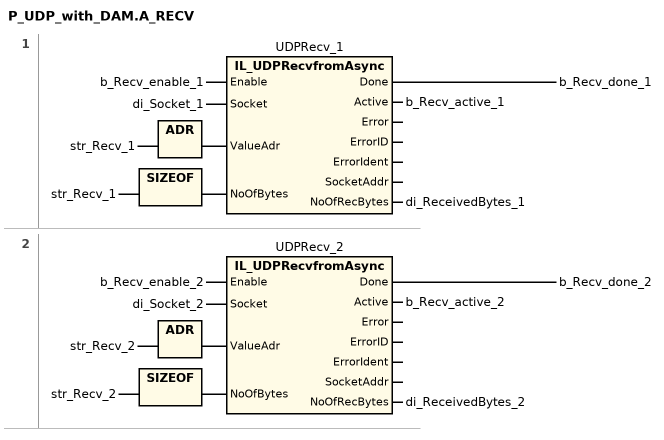
// NETWORK 1
UDPRecv_1(
    Enable := b_Recv_enable_1,
    Socket := di_Socket_1,
    ValueAdr := ADR(str_Recv_1),
    NoOfBytes := SIZEOF(str_Recv_1),
    Active => b_Recv_active_1,
    NoOfRecBytes => di_ReceivedBytes_1); // IL_UDPRecvfromAsync
b_Recv_done_1 := UDPRecv_1.Done;

// NETWORK 2
UDPRecv_2(
    Enable := b_Recv_enable_2,
    Socket := di_Socket_2,
    ValueAdr := ADR(str_Recv_2),
    NoOfBytes := SIZEOF(str_Recv_2),
    Active => b_Recv_active_2,
    NoOfRecBytes => di_ReceivedBytes_2); // IL_UDPRecvfromAsync
b_Recv_done_2 := UDPRecv_2.Done;
END_ACTION

ACTION A_SEND:
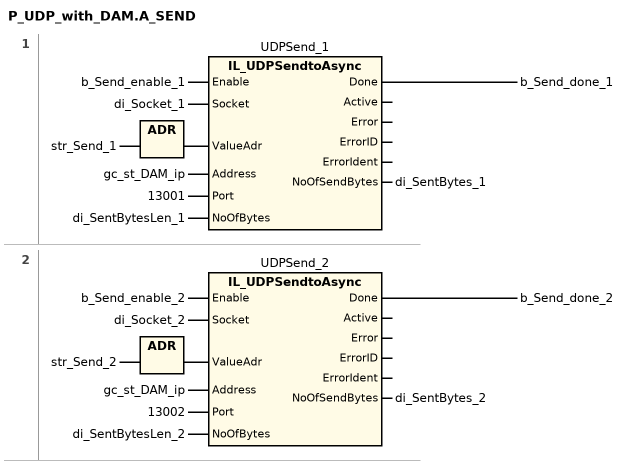
// NETWORK 1
UDPSend_1(
    Enable := b_Send_enable_1,
    Socket := di_Socket_1,
    ValueAdr := ADR(str_Send_1),
    Address := gc_st_DAM_ip,
    Port := 13001,
    NoOfBytes := di_SentBytesLen_1,
    NoOfSendBytes => di_SentBytes_1); // IL_UDPSendtoAsync
b_Send_done_1 := UDPSend_1.Done;

// NETWORK 2
UDPSend_2(
    Enable := b_Send_enable_2,
    Socket := di_Socket_2,
    ValueAdr := ADR(str_Send_2),
    Address := gc_st_DAM_ip,
    Port := 13002,
    NoOfBytes := di_SentBytesLen_2,
    NoOfSendBytes => di_SentBytes_2); // IL_UDPSendtoAsync
b_Send_done_2 := UDPSend_2.Done;
END_ACTION

END_PROGRAM

// IndraMotionMlc1/Application/POUs/TCP/Message/CRC16_MODBUS
FUNCTION_BLOCK CRC16_MODBUS
VAR_INPUT
	str_Message: ARRAY[1..40] OF BYTE;
	str_Len: BYTE;
END_VAR
VAR_OUTPUT
	crc16 : WORD;
END_VAR
VAR
	i : BYTE;
	j : BYTE;
	polynomial : WORD;
	curval : WORD;
	temp : WORD;
END_VAR


temp := 16#FFFF;
polynomial := 16#A001;
FOR i:=1 TO str_Len BY 1 DO
	curval := BYTE_TO_WORD(str_Message[i]);
	FOR j:=1 TO 8 BY 1 DO
		IF ((WORD_TO_BYTE(temp XOR curval) AND 16#01) = 16#01) THEN
			temp := (SHR(temp,1) XOR polynomial);
		ELSE
			temp := SHR(temp,1);			
		END_IF;
		curval := SHR(curval,1);
	END_FOR;
END_FOR;

crc16 := temp;

END_FUNCTION_BLOCK

// IndraMotionMlc1/Application/POUs/TCP/P_GSTAT_K2STAT
(*the program is built for GSTAT and KSTAT,according to ICD*)
PROGRAM P_GSTAT_K2STAT
VAR
(*the transitional variables for GSTAT and KSTAT*)
    STR_GSTAT: STRING(1500);
	STR_K2STAT: STRING(255);
	STR_K4STAT: STRING(255);

(*The function block BLINK generates a pulsating signal.The input consists of ENABLE of the type BOOL, as well as TIMELOW and TIMEHIGH of the type TIME.*)
	fb_blink_diagnos_1: BLINK;
	fb_blink_diagnos_2: BLINK;
	fb_blink_diagnos_3: BLINK;
	fb_blink_diagnos_4: BLINK;
	fb_blink_diagnos_5: BLINK;
	fb_blink_diagnos_6: BLINK;
	fb_blink_diagnos_MLC: BLINK;
(*With the function block "MB_ReadParameter" it is possible to read the current value of a parameter. The return value is DINT*)
	fb_read_brake_1: MB_ReadParameter;
	fb_read_brake_2: MB_ReadParameter;
	fb_read_brake_3: MB_ReadParameter;
	fb_read_brake_4: MB_ReadParameter;
	fb_read_brake_5: MB_ReadParameter;
	fb_read_brake_6: MB_ReadParameter;
(*With the function block "MB_ReadStringParameter" it is possible to read a parameter the operating data of which has the ASCII format (string).*)
	fb_diagnose_1: MB_ReadStringParameter;
	fb_diagnose_2: MB_ReadStringParameter;
	fb_diagnose_3: MB_ReadStringParameter;
	fb_diagnose_4: MB_ReadStringParameter;
	fb_diagnose_5: MB_ReadStringParameter;
	fb_diagnose_6: MB_ReadStringParameter;
	fb_diagnose_MLC: MB_ReadStringParameter;
(*With the function block "MB_ReadRealParameter" it is possible to read the current value of a parameter. The return value is REAL. *)
	FB_readcur1: MB_ReadRealParameter;
	FB_readcur2: MB_ReadRealParameter;
	FB_readcur3: MB_ReadRealParameter;
	FB_readcur4: MB_ReadRealParameter;
	FB_readcur5: MB_ReadRealParameter;
	FB_readcur6: MB_ReadRealParameter;
	fb_temp_1: MB_ReadRealParameter;
	fb_temp_2: MB_ReadRealParameter;
	fb_temp_3: MB_ReadRealParameter;
	fb_temp_4: MB_ReadRealParameter;
	fb_temp_5: MB_ReadRealParameter;
	fb_temp_6: MB_ReadRealParameter;
	fb_read_s189_1: MB_ReadRealParameter;
	fb_read_s189_3: MB_ReadRealParameter;
	fb_read_s189_5: MB_ReadRealParameter;
	FB_readtor1: MB_ReadRealParameter;
	FB_readtor2: MB_ReadRealParameter;
	FB_readtor3: MB_ReadRealParameter;
	FB_readtor4: MB_ReadRealParameter;
	FB_readtor5: MB_ReadRealParameter;
	FB_readtor6: MB_ReadRealParameter;
	FB_temp_1_a: MB_ReadRealParameter;
	FB_temp_2_a: MB_ReadRealParameter;
	FB_temp_3_a: MB_ReadRealParameter;
	FB_temp_4_a: MB_ReadRealParameter;
	FB_temp_5_a: MB_ReadRealParameter;
	FB_temp_6_a: MB_ReadRealParameter;
(*FP_P_0_0539,Holding brake status word *)
	dw_brake_1: DWORD;
	dw_brake_2: DWORD;
	dw_brake_3: DWORD;
	dw_brake_4: DWORD;
	dw_brake_5: DWORD;
	dw_brake_6: DWORD;
(*FP_P_0_0007,Display text of diagnostic message*)
	str_diagnose_MLC: STRING;
	str_diagnose_1: STRING;
	str_diagnose_2: STRING;
	str_diagnose_3: STRING;
	str_diagnose_4: STRING;
	str_diagnose_5: STRING;
	str_diagnose_6: STRING;

(*FP_S_0_0384,Amplifier temperature*)
	r_temp_amp1: REAL;
	r_temp_amp2: REAL;
	r_temp_amp3: REAL;
	r_temp_amp4: REAL;
	r_temp_amp5: REAL;
	r_temp_amp6: REAL;


(*<<<<<<<<<<<<<<<<<<<<<<<<<<<<<<<<<<<<<<<add MLC temperature and operation hour(20100708)>>>>>>>>>>>>>>>>>>>>>>>>>>>>>>>>>>>>>*)
	fb_temp_MLC: MB_ReadRealParameter;
	r_temp_MLC: REAL;(*FP_c_0_0070,Control unit temperature*)
	fb_read_system_status: MB_ReadParameter;
	dw_system_status: DWORD;(*FP_C_0_0023,MC system status,used for temperature warning*)
	fb_read_operation_hour: MB_ReadParameter;

(*the limit for judging whether azimuth following error is too big*)
	r_limit_track_az: REAL;
(*test for limit check*)
	fb_software_limit_1: MB_ReadParameter;
	fb_software_limit_5: MB_ReadParameter;
	fb_software_limit_3: MB_ReadParameter;
	fb_hardware_limit_1: MB_ReadParameter;
	fb_hardware_limit_3: MB_ReadParameter;
	fb_hardware_limit_5: MB_ReadParameter;
	fb_ESTOP_1: MB_ReadParameter;
	fb_ESTOP_3: MB_ReadParameter;
	fb_ESTOP_5: MB_ReadParameter;
	i_software_limit_1: DINT;
	i_software_limit_3: DINT;
	i_software_limit_5: DINT;
	i_hardware_limit_1: DINT;
	i_hardware_limit_3: DINT;
	i_hardware_limit_5: DINT;
	i_ESTOP_1: DINT;
	i_ESTOP_3: DINT;
	i_ESTOP_5: DINT;


	b_azimuth_limit: BOOL;
	b_elevation_limit: BOOL;
	b_FeedIndexer_limit: BOOL;
	fb_readpar_speed_1: MB_ReadRealParameter;
	fb_readpar_speed_3: MB_ReadRealParameter;
	fb_readpar_speed_5: MB_ReadRealParameter;
	
	str_concat: ARRAY[1..40] OF STRING(1500);(*数组及其类型的定义*)	
	Counter: INT;
	FB_readmotorencoder1: MB_ReadRealParameter;
	FB_readmotorencoder2: MB_ReadRealParameter;
	FB_readmotorencoder3: MB_ReadRealParameter;
	FB_readmotorencoder4: MB_ReadRealParameter;
	FB_readmotorencoder5: MB_ReadRealParameter;
	FB_readmotorencoder6: MB_ReadRealParameter;
	r_motorencoder_6: REAL;
	r_motorencoder_5: REAL;
	r_motorencoder_4: REAL;
	r_motorencoder_3: REAL;
	r_motorencoder_2: REAL;
	r_motorencoder_1: REAL;
	
	(*the status word for GSTAT*)
	
	status_1:DWORD;
	status_2:DWORD;
	status_3:DWORD;
	status_4:DWORD;
	status_5:DWORD;
	status_6:DWORD;
	fb_diagnose_111: MB_ReadParameter;
	str_diagnose_11: DWORD;
	fb_blink_diagnos_11: BLINK;
	fb_diagnose_11: MB_ReadrealParameter;
	str_diagnose_111: REAL;
	fb_readpar_speed_2: MB_ReadRealParameter;
	fb_readpar_speed_4: MB_ReadRealParameter;
	fb_readpar_speed_6: MB_ReadRealParameter;
	
	ReadAxisPshape: ARRAY[1..5] OF MB_ReadlrealParameter;
	ReadAxisVact: ARRAY[1..5] OF MB_ReadlrealParameter;
	ReadAxisVshape: ARRAY[1..5] OF MB_ReadlrealParameter;

	conut_i: INT;
	b_PID_in_FI: BOOL;
	b_limit_cw_FI: BOOL;
	b_limit_ccw_FI: BOOL;
	b_limit_final_FI: BOOL;
	fb_readpar_pos_cmd_1: MB_ReadRealParameter;
END_VAR

P_GSTAT_K2STAT.A_Read_Parameter();

status_code1:=LEFT(str_diagnose_1,5);
status_code2:=LEFT(str_diagnose_2,5);
status_code3:=LEFT(str_diagnose_3,5);
status_code4:=LEFT(str_diagnose_4,5);
status_code5:=LEFT(str_diagnose_5,5);
status_code6:=LEFT(str_diagnose_6,5);

FOR  conut_i:=1 TO 5 BY 1 DO
ReadAxisPshape[conut_i](
	Enable:=axisdata[1].Axis_Inbb , 
	Done=> , 
	Active=> , 
	Error=> , 
	ErrorID=> , 
	ErrorIdent=> , 
	ParameterNumber:=FP_P_0_0434 , 
	Value=>P_shape_value[conut_i] , 
	Axis:=AxRef[conut_i] );
	
ReadAxisVshape[conut_i](
	Enable:=axisdata[1].Axis_Inbb , 
	Done=> , 
	Active=> , 
	Error=> , 
	ErrorID=> , 
	ErrorIdent=> , 
	ParameterNumber:=FP_P_0_0434 , 
	Value=>V_shape_value[conut_i] , 
	Axis:=AxRef[conut_i] );
	
ReadAxisVact[conut_i](
	Enable:=axisdata[1].Axis_Inbb , 
	Done=> , 
	Active=> , 
	Error=> , 
	ErrorID=> , 
	ErrorIdent=> , 
	ParameterNumber:=FP_S_0_0040 , 
	Value=>V_act_value[conut_i] , 
	Axis:=AxRef[conut_i] );
END_FOR

(*<<<<<<<<<<<<<<<<<<<<<<<<<<<<<master_status>>>>>>>>>>>>>>>>>>>>>>>>>>>>>>>>>>>>>>>>>>>>>>>>>>>>>>>*)
master_status.0:=axisdata[1].Axis_InAb;
IF b_remote_on=TRUE THEN
	master_status.1:=0;
ELSE
	master_status.1:=1;
END_IF
IF b_DSdoor_Estop  THEN
	master_status.2:=1;
ELSE
	master_status.2:=0;
END_IF

IF ABS(axisdata[3].rActualPosition_i-90)<0.02 THEN
	master_status.3:=1;
ELSE
	master_status.3:=0;
END_IF
	master_status.4:=(axisdata[1].Axis_Error OR axisdata[2].Axis_Error OR axisdata[3].Axis_Error OR axisdata[4].Axis_Error OR axisdata[5].Axis_Error OR axisdata[6].Axis_Error);
	master_status.5:=b_stow_pin_limit_unlock;
	master_status.6:=b_stow_pin_limit_lock;
	
IF i_num_stack_left>9500 THEN
		master_status.7:=0;
	ELSE IF i_num_stack_left<1500 THEN
		master_status.7:=1;	
	END_IF
		
END_IF

IF b_remote_on_run AND b_track_on THEN
	master_status.9:=0;
	master_status.8:=1;
ELSIF b_remote_on_run AND b_Track_Pause = TRUE THEN
	master_status.9:=1;
	master_status.8:=0;
ELSIF b_remote_on_run AND b_Track_Pause = FALSE  AND b_track_on = FALSE THEN
	master_status.9:=0;
	master_status.8:=0;
ELSE
 	master_status.9:=1;
	master_status.8:=1;
END_IF

IF 	b_encoder_ok_az	AND b_encoder_ok_FI THEN
	master_status.10:=1;
	master_status.11:=1;
ELSIF b_encoder_ok_az =FALSE AND b_encoder_ok_FI THEN
	master_status.10:=0;
	master_status.11:=1;
ELSIF b_encoder_ok_az  AND b_encoder_ok_FI=FALSE THEN
	master_status.10:=1;
	master_status.11:=0;
ELSE
	master_status.10:=0;
	master_status.11:=0;		
END_IF

IF b_remote_on_run THEN
	master_status.12:=1;
ELSE
	master_status.12:=0;
END_IF
	
IF b_remote_on_run THEN
	master_status.12:=1;
ELSE
	master_status.12:=0;
END_IF

IF b_permit_new_file THEN
	master_status.13:=1;
ELSE
	master_status.13:=0;
END_IF

(*<<<<<<<<<<<<<<<<<<<<<<<<<<<<<status_1>>>>>>>>>>>>>>>>>>>>>>>>>>>>>>>>>>>>>>>>>>>>>>>>>>>>>>>*)
status_1.0:=axisdata[1].Axis_InAb;
status_1.1:=b_PID_in_az;
status_1.2:=dw_brake_1.0;
status_1.3:=b_limit_cw_az;
status_1.4:=b_limit_ccw_az;
status_1.5:=(b_limit_final_cw_az OR b_limit_final_ccw_az);
status_1.6:=axisdata[1].Axis_Error;

(*<<<<<<<<<<<<<<<<<<<<<<<<<<<<<status_2>>>>>>>>>>>>>>>>>>>>>>>>>>>>>>>>>>>>>>>>>>>>>>>>>>>>>>>*)
status_2.0:=axisdata[2].Axis_InAb;
status_2.1:=b_PID_in_az;
status_2.2:=dw_brake_2.0;
status_2.3:=b_limit_cw_az;
status_2.4:=b_limit_ccw_az;
status_2.5:=(b_limit_final_cw_az OR b_limit_final_ccw_az);
status_2.6:=axisdata[2].Axis_Error;

(*<<<<<<<<<<<<<<<<<<<<<<<<<<<<<status_3>>>>>>>>>>>>>>>>>>>>>>>>>>>>>>>>>>>>>>>>>>>>>>>>>>>>>>>*)
status_3.0:=axisdata[3].Axis_InAb;
status_3.1:=b_PID_in_el;
status_3.2:=dw_brake_3.0;
status_3.3:=b_limit_cw_el;
status_3.4:=b_limit_ccw_el;
status_3.5:=(b_limit_final_cw_el OR b_limit_final_ccw_el) ;
status_3.6:=axisdata[3].Axis_Error;

(*<<<<<<<<<<<<<<<<<<<<<<<<<<<<<status_4>>>>>>>>>>>>>>>>>>>>>>>>>>>>>>>>>>>>>>>>>>>>>>>>>>>>>>>*)
status_4.0:=axisdata[4].Axis_InAb;
status_4.1:=b_PID_in_el;
status_4.2:=dw_brake_4.0;
status_4.3:=b_limit_cw_el;
status_4.4:=b_limit_ccw_el;
status_4.5:=(b_limit_final_cw_el OR b_limit_final_ccw_el); 
status_4.6:=axisdata[4].Axis_Error;

(*<<<<<<<<<<<<<<<<<<<<<<<<<<<<<status_5>>>>>>>>>>>>>>>>>>>>>>>>>>>>>>>>>>>>>>>>>>>>>>>>>>>>>>>*)
status_5.0:=axisdata[5].Axis_InAb;
status_5.1:=b_PID_in_FI;
status_5.2:=dw_brake_5.0;
status_5.3:=b_limit_cw_FI;
status_5.4:=b_limit_ccw_FI;
status_5.5:=b_limit_final_FI;
status_5.6:=axisdata[5].Axis_Error;

(*<<<<<<<<<<<<<<<<<<<<<<<<<<<<<status_6>>>>>>>>>>>>>>>>>>>>>>>>>>>>>>>>>>>>>>>>>>>>>>>>>>>>>>>*)
status_6.0:=axisdata[6].Axis_InAb;
status_6.1:=b_PID_in_FI;
status_6.2:=dw_brake_6.0;
status_6.3:=b_limit_cw_FI;
status_6.4:=b_limit_ccw_FI;
status_6.5:=b_limit_final_FI;
status_6.6:=axisdata[6].Axis_Error;


(*
(*<<<<<<<<<<<<<<<<<<<<<<<<<<<<<status_2>>>>>>>>>>>>>>>>>>>>>>>>>>>>>>>>>>>>>>>>>>>>>>>>>>>>>>>*)
status_2.0:=NOT(axisdata[2].Axis_InAb);
status_2.1:=axisdata[2].Axis_Error;
status_2.2:=NOT(dw_brake_2.0);
IF r_temp_motor2>120 THEN
status_2.3:=1;
b_power_Az:=FALSE;
b_enable_az_1:=FALSE;
b_enable_az_2:=FALSE;
ELSE
status_2.3:=0;
END_IF
IF r_current_2>5 THEN
status_2.4:=1;
ELSE
status_2.4:=0;
END_IF
(*<<<<<<<<<<<<<<<<<<<<<<<<<<<<<status_3>>>>>>>>>>>>>>>>>>>>>>>>>>>>>>>>>>>>>>>>>>>>>>>>>>>>>>>*)
status_3.0:=NOT(axisdata[3].Axis_InAb);
status_3.1:=axisdata[3].Axis_Error;
status_3.2:=NOT(dw_brake_3.0);
IF r_temp_motor3>120 THEN
status_3.3:=1;
b_power_El:=FALSE;
b_enable_el_3:=FALSE;
b_enable_el_4:=FALSE;
ELSE
status_3.3:=0;
END_IF
IF r_current_3>5 THEN
status_3.4:=1;
ELSE
status_3.4:=0;
END_IF
status_3.8:=NOT(b_PID_in_el);

IF (b_scc_goto=TRUE AND (b_goto_Az_done=FALSE OR b_goto_El_done=FALSE OR b_goto_FI_done=FALSE)) OR (b_track_on=TRUE AND i_num_stack_left<>0) THEN
status_3.9:=1;
END_IF;
IF (b_goto_Az_done=TRUE AND b_goto_El_done=TRUE AND b_goto_FI_done=TRUE) OR i_num_stack_left=0 THEN
status_3.9:=0;
END_IF;

status_3.10:=NOT(b_track_on);
IF ABS(r_track_error[2])<0.0034 THEN
	status_3.11:=0;
ELSE
	status_3.11:=1;
END_IF
status_3.12:=axisdata[3].Axis_Error;
IF ABS(r_following_3)>0.5 THEN
status_3.13:=1;
ELSE
status_3.13:=0;
END_IF
IF r_pos_el<14.6 THEN
	status_3.14:=1;
ELSE
	status_3.14:=0;
END_IF
IF r_pos_el>90.15 THEN
	status_3.15:=1;
ELSE
	status_3.15:=0;
END_IF
status_3.16:=b_limit_ccw_el;
status_3.17:=b_limit_cw_el;
status_3.18:=b_limit_final_el;
status_3.19:=b_track_overspeed_el;
(*<<<<<<<<<<<<<<<<<<<<<<<<<<<<<status_4>>>>>>>>>>>>>>>>>>>>>>>>>>>>>>>>>>>>>>>>>>>>>>>>>>>>>>>*)
status_4.0:=NOT(axisdata[4].Axis_InAb);
status_4.1:=axisdata[4].Axis_Error;
status_4.2:=NOT(dw_brake_4.0);
IF r_temp_motor4>120 THEN
status_4.3:=1;
b_power_El:=FALSE;
b_enable_el_3:=FALSE;
b_enable_el_4:=FALSE;
ELSE
status_4.3:=0;
END_IF
IF r_current_4>5 THEN
status_4.4:=1;
ELSE
status_4.4:=0;
END_IF
(*<<<<<<<<<<<<<<<<<<<<<<<<<<<<<status_5>>>>>>>>>>>>>>>>>>>>>>>>>>>>>>>>>>>>>>>>>>>>>>>>>>>>>>>*)
status_5.0:=NOT(axisdata[5].Axis_InAb);
status_5.1:=axisdata[5].Axis_Error;
status_5.2:=NOT(dw_brake_5.0);
IF r_temp_motor5>120 THEN
status_5.3:=1;
b_power_FI:=FALSE;
b_enable_FI_5:=FALSE;
ELSE
status_5.3:=0;
END_IF
IF r_current_5>5 THEN
status_5.4:=1;
ELSE
status_5.4:=0;
END_IF

status_5.8:=NOT(b_gearinpos_5_done);

IF (b_scc_goto=TRUE AND (b_goto_Az_done=FALSE OR b_goto_El_done=FALSE OR b_goto_FI_done=FALSE)) OR (b_track_on=TRUE AND i_num_stack_left<>0) THEN
status_5.9:=1;
END_IF;
IF (b_goto_Az_done=TRUE AND b_goto_El_done=TRUE AND b_goto_FI_done=TRUE) OR i_num_stack_left=0 THEN
status_5.9:=0;
END_IF;

status_5.10:=NOT(b_track_on);
IF ABS(r_track_error[3])<0.0034 THEN
	status_5.11:=0;
ELSE
	status_5.11:=1;
END_IF
status_5.12:=axisdata[5].Axis_Error;
IF ABS(r_following_5)>0.5 THEN
status_5.13:=1;
ELSE
status_5.13:=0;
END_IF

IF r_pos_FI<-89 THEN
	status_5.14:=1;
ELSE
	status_5.14:=0;
END_IF

IF r_pos_FI>89 THEN
	status_5.15:=1;
ELSE
	status_5.15:=0;
END_IF
status_5.16:=b_limit_ccw_FI;
status_5.17:=b_limit_cw_FI;
status_5.18:=b_limit_final_FI;
status_5.19:=b_track_overspeed_FI;
*)

(*<<<<<<<<<<<<<<<<<<<<<<<<<<<<<concatenate STR_GSTAT>>>>>>>>>>>>>>>>>>>>>>>>>>>>>>>>>>>>>>>>>>>>>>>>>>>>>>>*)
str_concat[1]:=CONCAT(' ',DWORD_TO_STRING(status_1));
str_concat[2]:=CONCAT(' ',LREAL_TO_STRING(F_reduce_to_1_bit(LREAL_TO_STRING(r_current_1))));
str_concat[3]:=CONCAT(' ',LREAL_TO_STRING(r_temp_motor1));
str_concat[4]:=CONCAT(' ',LREAL_TO_STRING(i_speed_1));
str_concat[5]:=CONCAT(' ',LREAL_TO_STRING(F_reduce_to_1_bit(LREAL_TO_STRING(r_motorencoder_1))));


str_concat[6]:=CONCAT(' ',DWORD_TO_STRING(status_2));
str_concat[7]:=CONCAT(' ',LREAL_TO_STRING(F_reduce_to_1_bit(LREAL_TO_STRING(r_current_2))));
str_concat[8]:=CONCAT(' ',LREAL_TO_STRING(r_temp_motor2));
str_concat[9]:=CONCAT(' ',LREAL_TO_STRING(i_speed_2));
str_concat[10]:=CONCAT(' ',LREAL_TO_STRING(F_reduce_to_1_bit(LREAL_TO_STRING(r_motorencoder_2))));

str_concat[11]:=CONCAT(' ',DWORD_TO_STRING(status_3));
str_concat[12]:=CONCAT(' ',LREAL_TO_STRING(F_reduce_to_1_bit(LREAL_TO_STRING(r_current_3))));
str_concat[13]:=CONCAT(' ',LREAL_TO_STRING(r_temp_motor3));
str_concat[14]:=CONCAT(' ',LREAL_TO_STRING(i_speed_3));
str_concat[15]:=CONCAT(' ',LREAL_TO_STRING(F_reduce_to_1_bit(LREAL_TO_STRING(r_motorencoder_3))));

str_concat[16]:=CONCAT(' ',DWORD_TO_STRING(status_4));
str_concat[17]:=CONCAT(' ',LREAL_TO_STRING(F_reduce_to_1_bit(LREAL_TO_STRING(r_current_4))));
str_concat[18]:=CONCAT(' ',LREAL_TO_STRING(r_temp_motor4));
str_concat[19]:=CONCAT(' ',LREAL_TO_STRING(i_speed_4));
str_concat[20]:=CONCAT(' ',LREAL_TO_STRING(F_reduce_to_1_bit(LREAL_TO_STRING(r_motorencoder_4))));

str_concat[21]:=CONCAT(' ',DWORD_TO_STRING(status_5));
str_concat[22]:=CONCAT(' ',LREAL_TO_STRING(F_reduce_to_1_bit(LREAL_TO_STRING(r_current_5))));
str_concat[23]:=CONCAT(' ',LREAL_TO_STRING(r_temp_motor5));
str_concat[24]:=CONCAT(' ',LREAL_TO_STRING(i_speed_5));
str_concat[25]:=CONCAT(' ',LREAL_TO_STRING(F_reduce_to_1_bit(LREAL_TO_STRING(r_motorencoder_5))));

str_concat[26]:=CONCAT(' ',DWORD_TO_STRING(status_6));
str_concat[27]:=CONCAT(' ',LREAL_TO_STRING(F_reduce_to_1_bit(LREAL_TO_STRING(r_current_6))));
str_concat[28]:=CONCAT(' ',LREAL_TO_STRING(r_temp_motor6));
str_concat[29]:=CONCAT(' ',LREAL_TO_STRING(i_speed_6));
str_concat[30]:=CONCAT(' ',LREAL_TO_STRING(F_reduce_to_1_bit(LREAL_TO_STRING(r_motorencoder_6))));

str_concat[31]:=CONCAT(' ',last_command);
str_concat[32]:=CONCAT(' ',INT_TO_STRING(i_receive_cmd));
str_concat[33]:=CONCAT(' ',INT_TO_STRING(i_excute_cmd));
(*
str_concat[31]:=CONCAT(' ',REAL_TO_STRING(F_reduce_to_4_bit(REAL_TO_STRING(r_test1))));
str_concat[32]:=CONCAT(' ',REAL_TO_STRING(F_reduce_to_4_bit(REAL_TO_STRING(r_test2))));
str_concat[33]:=CONCAT(' ',REAL_TO_STRING(F_reduce_to_4_bit(REAL_TO_STRING(r_test3))));
*)
STR_GSTAT_M:='';(*for语句格式*)
				FOR Counter:=1 TO 33 BY 1 DO
					STR_GSTAT_M:=CONCAT(STR_GSTAT_M,str_concat[Counter]);
				END_FOR;



(*
STR_GSTAT:=CONCAT(STR_GSTAT,CONCAT(' ',DWORD_TO_STRING(status_1)));
STR_GSTAT:=CONCAT(STR_GSTAT,CONCAT(' ',REAL_TO_STRING(r_current_1)));
STR_GSTAT:=CONCAT(STR_GSTAT,CONCAT(' ',REAL_TO_STRING(r_temp_motor1)));
STR_GSTAT:=CONCAT(STR_GSTAT,CONCAT(' ',REAL_TO_STRING(i_speed_1)));
*)


(*
STR_GSTAT:=CONCAT(STR_GSTAT,CONCAT(' ',DWORD_TO_STRING(status_2)));
STR_GSTAT:=CONCAT(STR_GSTAT,CONCAT(' ',REAL_TO_STRING(r_current_2)));
STR_GSTAT:=CONCAT(STR_GSTAT,CONCAT(' ',REAL_TO_STRING(r_temp_motor2)));
STR_GSTAT:=CONCAT(STR_GSTAT,CONCAT(' ',REAL_TO_STRING(i_speed_1)));

STR_GSTAT:=CONCAT(STR_GSTAT,CONCAT(' ',DWORD_TO_STRING(status_3)));
STR_GSTAT:=CONCAT(STR_GSTAT,CONCAT(' ',REAL_TO_STRING(r_current_3)));
STR_GSTAT:=CONCAT(STR_GSTAT,CONCAT(' ',REAL_TO_STRING(r_temp_motor3)));
STR_GSTAT:=CONCAT(STR_GSTAT,CONCAT(' ',REAL_TO_STRING(i_speed_3)));

STR_GSTAT:=CONCAT(STR_GSTAT,CONCAT(' ',DWORD_TO_STRING(status_4)));
STR_GSTAT:=CONCAT(STR_GSTAT,CONCAT(' ',REAL_TO_STRING(r_current_4)));
STR_GSTAT:=CONCAT(STR_GSTAT,CONCAT(' ',REAL_TO_STRING(r_temp_motor4)));
STR_GSTAT:=CONCAT(STR_GSTAT,CONCAT(' ',REAL_TO_STRING(i_speed_3)));

STR_GSTAT:=CONCAT(STR_GSTAT,CONCAT(' ',DWORD_TO_STRING(status_5)));
STR_GSTAT:=CONCAT(STR_GSTAT,CONCAT(' ',REAL_TO_STRING(r_current_5)));
STR_GSTAT:=CONCAT(STR_GSTAT,CONCAT(' ',REAL_TO_STRING(r_temp_motor5)));
STR_GSTAT:=CONCAT(STR_GSTAT,CONCAT(' ',REAL_TO_STRING(i_speed_5)));

STR_GSTAT:=CONCAT(STR_GSTAT,CONCAT(' ',DWORD_TO_STRING(status_6)));
STR_GSTAT:=CONCAT(STR_GSTAT,CONCAT(' ',REAL_TO_STRING(r_current_6)));
STR_GSTAT:=CONCAT(STR_GSTAT,CONCAT(' ',REAL_TO_STRING(r_temp_motor6)));
STR_GSTAT:=CONCAT(STR_GSTAT,CONCAT(' ',REAL_TO_STRING(i_speed_5)));

STR_GSTAT:=CONCAT(STR_GSTAT,CONCAT(' ',INT_TO_STRING(i_num_stack_left)));
STR_GSTAT:=CONCAT(STR_GSTAT,CONCAT(' ',INT_TO_STRING(i_start)));
STR_GSTAT_M:=CONCAT(STR_GSTAT,CONCAT(' ',INT_TO_STRING(i_end)));

*)
(*<<<<<<<<<<<<<<<<<<<<<<<<<<<<<concatenate STR_K2STAT>>>>>>>>>>>>>>>>>>>>>>>>>>>>>>>>>>>>>>>>>>>>>>>>>>>>>>>*)
STR_K2STAT:=CONCAT('OK - ',REAL_TO_STRING(r_operation_hour/100));
STR_K2STAT:=CONCAT(STR_K2STAT,CONCAT(' ',LREAL_TO_STRING(r_temp_motor1)));
STR_K2STAT:=CONCAT(STR_K2STAT,CONCAT(' ',LREAL_TO_STRING(r_temp_motor2)));
STR_K2STAT:=CONCAT(STR_K2STAT,CONCAT(' ',LREAL_TO_STRING(r_temp_motor3)));
STR_K2STAT:=CONCAT(STR_K2STAT,CONCAT(' ',LREAL_TO_STRING(r_temp_motor4)));
STR_K2STAT:=CONCAT(STR_K2STAT,CONCAT(' ',LREAL_TO_STRING(r_temp_motor5)));
STR_K2STAT:=CONCAT(STR_K2STAT,CONCAT(' ',LREAL_TO_STRING(r_temp_amp1)));
STR_K2STAT:=CONCAT(STR_K2STAT,CONCAT(' ',LREAL_TO_STRING(r_temp_amp2)));
STR_K2STAT:=CONCAT(STR_K2STAT,CONCAT(' ',LREAL_TO_STRING(r_temp_amp3)));
STR_K2STAT:=CONCAT(STR_K2STAT,CONCAT(' ',LREAL_TO_STRING(r_temp_amp4)));
STR_K2STAT:=CONCAT(STR_K2STAT,CONCAT(' ',LREAL_TO_STRING(r_temp_amp5)));
STR_K2STAT_M:=CONCAT(STR_K2STAT,CONCAT(' ',LREAL_TO_STRING(r_temp_MLC)));
(*<<<<<<<<<<<<<<<<<<<<<<<<<<<<<concatenate STR_K4STAT>>>>>>>>>>>>>>>>>>>>>>>>>>>>>>>>>>>>>>>>>>>>>>>>>>>>>>>*)
STR_K4STAT:=CONCAT('OK - ',str_diagnose_MLC);
STR_K4STAT:=CONCAT(STR_K4STAT,CONCAT(' ',str_diagnose_1));
STR_K4STAT:=CONCAT(STR_K4STAT,CONCAT(' ',str_diagnose_2));
STR_K4STAT:=CONCAT(STR_K4STAT,CONCAT(' ',str_diagnose_3));
STR_K4STAT:=CONCAT(STR_K4STAT,CONCAT(' ',str_diagnose_4));
STR_K4STAT_M:=CONCAT(STR_K4STAT,CONCAT(' ',str_diagnose_5));

(*<<<<<<<<<<<<<<<<<<<<<<<<<<<<<concatenate STR_K5STAT>>>>>>>>>>>>>>>>>>>>>>>>>>>>>>>>>>>>>>>>>>>>>>>>>>>>>>>*)
IF i_software_limit_1=16 AND i_hardware_limit_1=3 AND i_ESTOP_1=5 THEN
	b_azimuth_limit:=TRUE;
ELSE
	b_azimuth_limit:=FALSE;
END_IF

IF i_software_limit_3=16 AND i_hardware_limit_3=3 AND i_ESTOP_3=5 THEN
	b_elevation_limit:=TRUE;
ELSE
	b_elevation_limit:=FALSE;
END_IF

IF i_software_limit_5=16 AND i_hardware_limit_5=3 AND i_ESTOP_5=5 THEN
	b_FeedIndexer_limit:=TRUE;
ELSE
	b_FeedIndexer_limit:=FALSE;
END_IF
IF b_azimuth_limit AND b_elevation_limit AND b_FeedIndexer_limit THEN
	STR_K5STAT_M:='All the axes are safe.';
ELSE
	STR_K5STAT_M:='';
	IF b_azimuth_limit=FALSE THEN
		STR_K5STAT_M:=CONCAT(STR_K5STAT_M,'Azimuth axis is unsafe. ');
	END_IF
	IF b_elevation_limit=FALSE THEN
		STR_K5STAT_M:=CONCAT(STR_K5STAT_M,'Elevation axis is unsafe. ');
	END_IF
	IF b_FeedIndexer_limit=FALSE THEN
		STR_K5STAT_M:=CONCAT(STR_K5STAT_M,'FeedIndexer axis is unsafe. ');
	END_IF
END_IF

ACTION A_Read_Parameter:
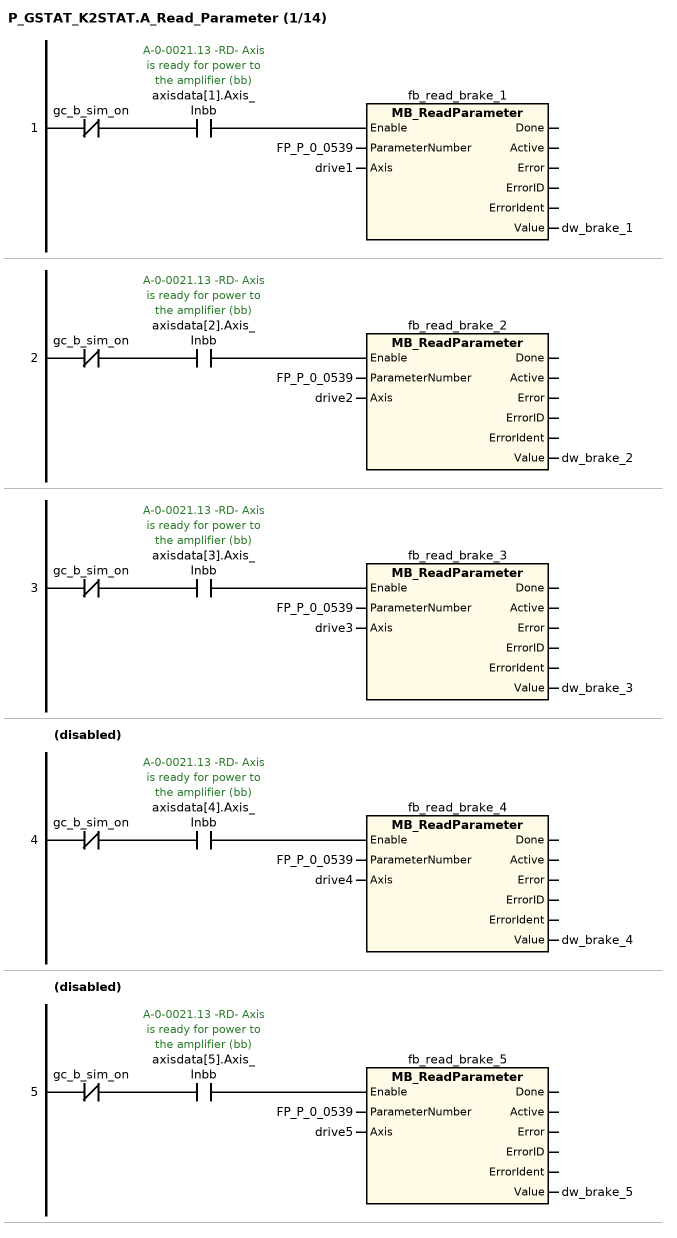
// NETWORK 1
//   fb_read_brake_1: With the function block "MB_ReadParameter" it is possible to read the current value of a parameter. The return value is DINT
//   axisdata[1].Axis_Inbb: A-0-0021.13 -RD- Axis is ready for power to the amplifier (bb)
//   FP_P_0_0539: Holding brake status word
//   drive1: Real axis "Drive1" with axis number 1
//   dw_brake_1: FP_P_0_0539,Holding brake status word
fb_read_brake_1(
    Enable := NOT gc_b_sim_on AND axisdata[1].Axis_Inbb,
    ParameterNumber := FP_P_0_0539,
    Axis := drive1,
    Value => dw_brake_1); // MB_ReadParameter

// NETWORK 2
//   axisdata[2].Axis_Inbb: A-0-0021.13 -RD- Axis is ready for power to the amplifier (bb)
//   FP_P_0_0539: Holding brake status word
//   drive2: Real axis "Drive2" with axis number 2
fb_read_brake_2(
    Enable := NOT gc_b_sim_on AND axisdata[2].Axis_Inbb,
    ParameterNumber := FP_P_0_0539,
    Axis := drive2,
    Value => dw_brake_2); // MB_ReadParameter

// NETWORK 3
//   axisdata[3].Axis_Inbb: A-0-0021.13 -RD- Axis is ready for power to the amplifier (bb)
//   FP_P_0_0539: Holding brake status word
//   drive3: Real axis "Drive3" with axis number 3
fb_read_brake_3(
    Enable := NOT gc_b_sim_on AND axisdata[3].Axis_Inbb,
    ParameterNumber := FP_P_0_0539,
    Axis := drive3,
    Value => dw_brake_3); // MB_ReadParameter

// NETWORK 4 (disabled)
//   axisdata[4].Axis_Inbb: A-0-0021.13 -RD- Axis is ready for power to the amplifier (bb)
//   FP_P_0_0539: Holding brake status word
//   drive4: Real axis "Drive4" with axis number 4
// fb_read_brake_4(
//     Enable := NOT gc_b_sim_on AND axisdata[4].Axis_Inbb,
//     ParameterNumber := FP_P_0_0539,
//     Axis := drive4,
//     Value => dw_brake_4); // MB_ReadParameter

// NETWORK 5 (disabled)
//   axisdata[5].Axis_Inbb: A-0-0021.13 -RD- Axis is ready for power to the amplifier (bb)
//   FP_P_0_0539: Holding brake status word
//   drive5: Real axis "Drive5" with axis number 5
// fb_read_brake_5(
//     Enable := NOT gc_b_sim_on AND axisdata[5].Axis_Inbb,
//     ParameterNumber := FP_P_0_0539,
//     Axis := drive5,
//     Value => dw_brake_5); // MB_ReadParameter

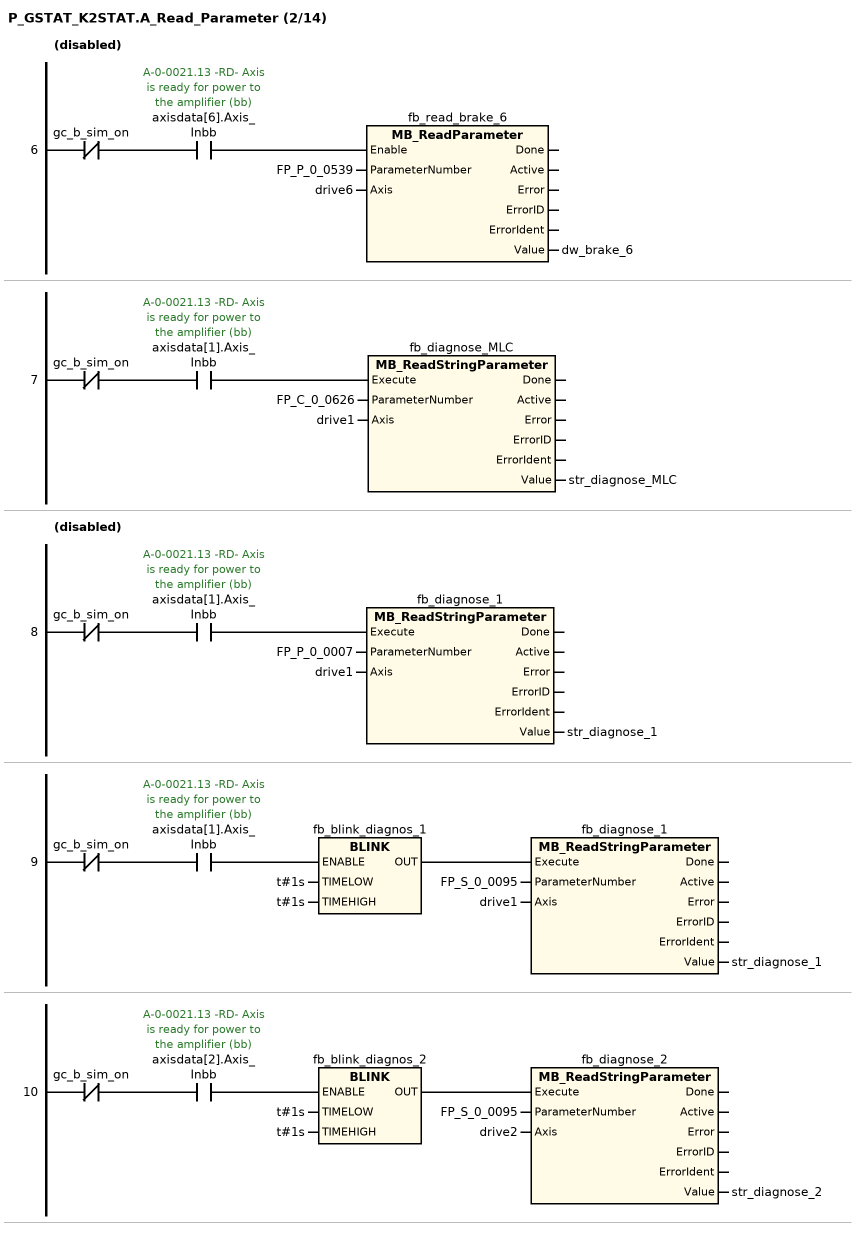
// NETWORK 6 (disabled)
//   axisdata[6].Axis_Inbb: A-0-0021.13 -RD- Axis is ready for power to the amplifier (bb)
//   FP_P_0_0539: Holding brake status word
//   drive6: Real axis "Drive6" with axis number 6
// fb_read_brake_6(
//     Enable := NOT gc_b_sim_on AND axisdata[6].Axis_Inbb,
//     ParameterNumber := FP_P_0_0539,
//     Axis := drive6,
//     Value => dw_brake_6); // MB_ReadParameter

// NETWORK 7
//   axisdata[1].Axis_Inbb: A-0-0021.13 -RD- Axis is ready for power to the amplifier (bb)
//   FP_C_0_0626: Diagnostics
//   drive1: Real axis "Drive1" with axis number 1
//   str_diagnose_MLC: FP_P_0_0007,Display text of diagnostic message
fb_diagnose_MLC(
    Execute := NOT gc_b_sim_on AND axisdata[1].Axis_Inbb,
    ParameterNumber := FP_C_0_0626,
    Axis := drive1,
    Value => str_diagnose_MLC); // MB_ReadStringParameter

// NETWORK 8 (disabled)
//   fb_diagnose_1: With the function block "MB_ReadStringParameter" it is possible to read a parameter the operating data of which has the ASCII format (string).
//   axisdata[1].Axis_Inbb: A-0-0021.13 -RD- Axis is ready for power to the amplifier (bb)
//   FP_P_0_0007: Display text of diagnostic message
//   drive1: Real axis "Drive1" with axis number 1
// fb_diagnose_1(
//     Execute := NOT gc_b_sim_on AND axisdata[1].Axis_Inbb,
//     ParameterNumber := FP_P_0_0007,
//     Axis := drive1,
//     Value => str_diagnose_1); // MB_ReadStringParameter

// NETWORK 9
//   fb_diagnose_1: With the function block "MB_ReadStringParameter" it is possible to read a parameter the operating data of which has the ASCII format (string).
//   fb_blink_diagnos_1: The function block BLINK generates a pulsating signal.The input consists of ENABLE of the type BOOL, as well as TIMELOW and TIMEHIGH of the type TIME.
//   axisdata[1].Axis_Inbb: A-0-0021.13 -RD- Axis is ready for power to the amplifier (bb)
//   FP_S_0_0095: Diagnostic message
//   drive1: Real axis "Drive1" with axis number 1
fb_blink_diagnos_1(ENABLE := NOT gc_b_sim_on AND axisdata[1].Axis_Inbb, TIMELOW := t#1s, TIMEHIGH := t#1s); // BLINK
fb_diagnose_1(
    Execute := fb_blink_diagnos_1.OUT,
    ParameterNumber := FP_S_0_0095,
    Axis := drive1,
    Value => str_diagnose_1); // MB_ReadStringParameter

// NETWORK 10
//   axisdata[2].Axis_Inbb: A-0-0021.13 -RD- Axis is ready for power to the amplifier (bb)
//   FP_S_0_0095: Diagnostic message
//   drive2: Real axis "Drive2" with axis number 2
fb_blink_diagnos_2(ENABLE := NOT gc_b_sim_on AND axisdata[2].Axis_Inbb, TIMELOW := t#1s, TIMEHIGH := t#1s); // BLINK
fb_diagnose_2(
    Execute := fb_blink_diagnos_2.OUT,
    ParameterNumber := FP_S_0_0095,
    Axis := drive2,
    Value => str_diagnose_2); // MB_ReadStringParameter

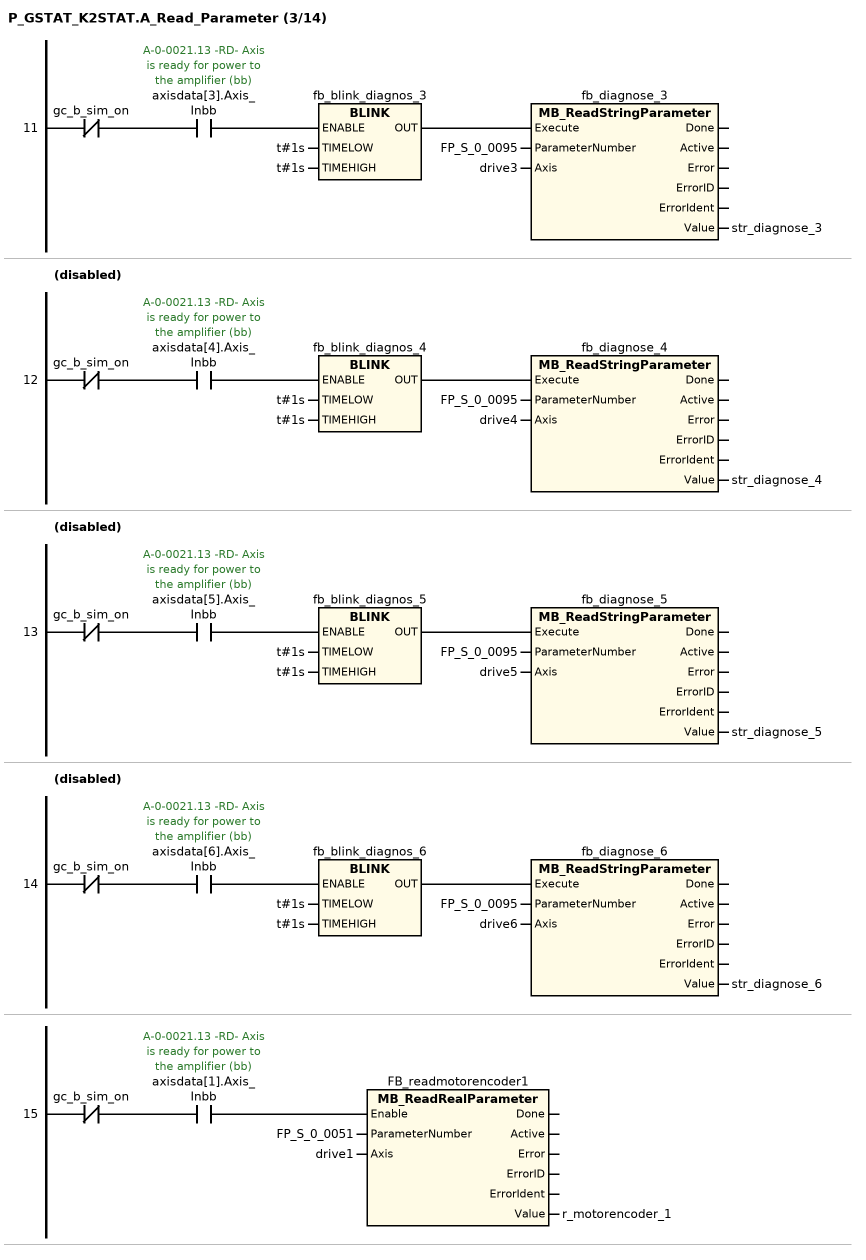
// NETWORK 11
//   axisdata[3].Axis_Inbb: A-0-0021.13 -RD- Axis is ready for power to the amplifier (bb)
//   FP_S_0_0095: Diagnostic message
//   drive3: Real axis "Drive3" with axis number 3
fb_blink_diagnos_3(ENABLE := NOT gc_b_sim_on AND axisdata[3].Axis_Inbb, TIMELOW := t#1s, TIMEHIGH := t#1s); // BLINK
fb_diagnose_3(
    Execute := fb_blink_diagnos_3.OUT,
    ParameterNumber := FP_S_0_0095,
    Axis := drive3,
    Value => str_diagnose_3); // MB_ReadStringParameter

// NETWORK 12 (disabled)
//   axisdata[4].Axis_Inbb: A-0-0021.13 -RD- Axis is ready for power to the amplifier (bb)
//   FP_S_0_0095: Diagnostic message
//   drive4: Real axis "Drive4" with axis number 4
// fb_blink_diagnos_4(ENABLE := NOT gc_b_sim_on AND axisdata[4].Axis_Inbb, TIMELOW := t#1s, TIMEHIGH := t#1s); // BLINK
// fb_diagnose_4(
//     Execute := fb_blink_diagnos_4.OUT,
//     ParameterNumber := FP_S_0_0095,
//     Axis := drive4,
//     Value => str_diagnose_4); // MB_ReadStringParameter

// NETWORK 13 (disabled)
//   axisdata[5].Axis_Inbb: A-0-0021.13 -RD- Axis is ready for power to the amplifier (bb)
//   FP_S_0_0095: Diagnostic message
//   drive5: Real axis "Drive5" with axis number 5
// fb_blink_diagnos_5(ENABLE := NOT gc_b_sim_on AND axisdata[5].Axis_Inbb, TIMELOW := t#1s, TIMEHIGH := t#1s); // BLINK
// fb_diagnose_5(
//     Execute := fb_blink_diagnos_5.OUT,
//     ParameterNumber := FP_S_0_0095,
//     Axis := drive5,
//     Value => str_diagnose_5); // MB_ReadStringParameter

// NETWORK 14 (disabled)
//   axisdata[6].Axis_Inbb: A-0-0021.13 -RD- Axis is ready for power to the amplifier (bb)
//   FP_S_0_0095: Diagnostic message
//   drive6: Real axis "Drive6" with axis number 6
// fb_blink_diagnos_6(ENABLE := NOT gc_b_sim_on AND axisdata[6].Axis_Inbb, TIMELOW := t#1s, TIMEHIGH := t#1s); // BLINK
// fb_diagnose_6(
//     Execute := fb_blink_diagnos_6.OUT,
//     ParameterNumber := FP_S_0_0095,
//     Axis := drive6,
//     Value => str_diagnose_6); // MB_ReadStringParameter

// NETWORK 15
//   axisdata[1].Axis_Inbb: A-0-0021.13 -RD- Axis is ready for power to the amplifier (bb)
//   FP_S_0_0051: Position feedback value 1
//   drive1: Real axis "Drive1" with axis number 1
FB_readmotorencoder1(
    Enable := NOT gc_b_sim_on AND axisdata[1].Axis_Inbb,
    ParameterNumber := FP_S_0_0051,
    Axis := drive1,
    Value => r_motorencoder_1); // MB_ReadRealParameter

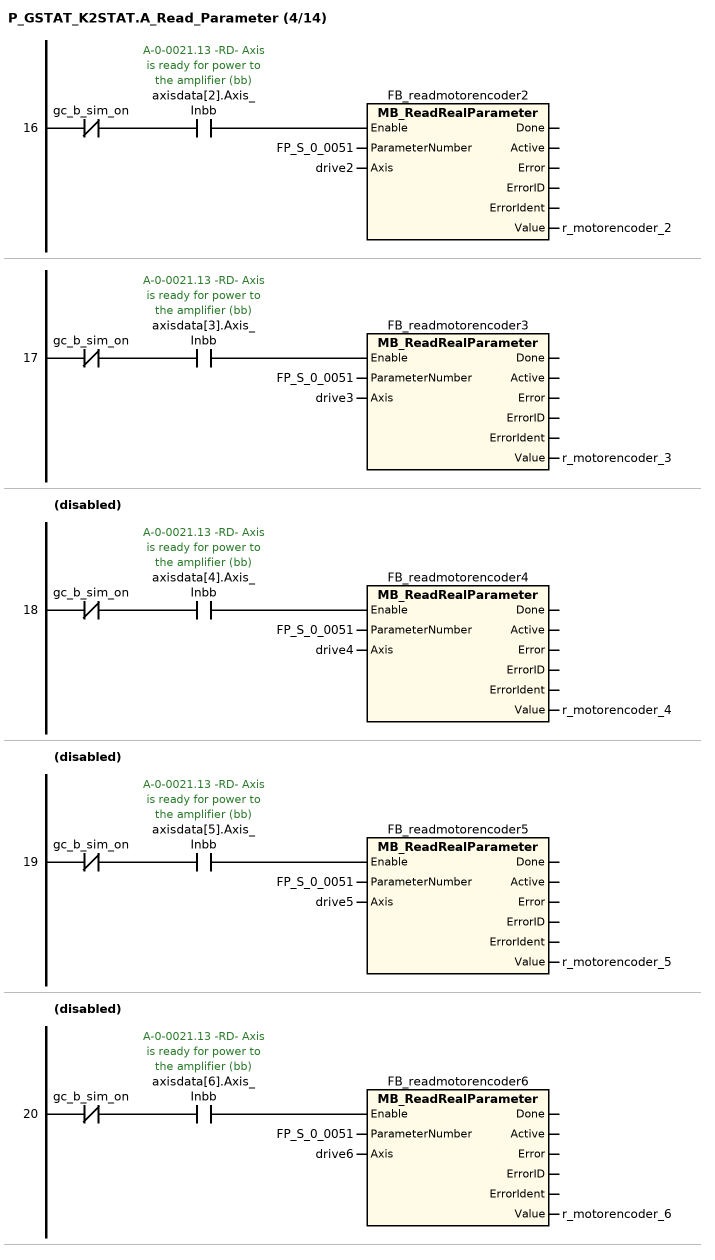
// NETWORK 16
//   axisdata[2].Axis_Inbb: A-0-0021.13 -RD- Axis is ready for power to the amplifier (bb)
//   FP_S_0_0051: Position feedback value 1
//   drive2: Real axis "Drive2" with axis number 2
FB_readmotorencoder2(
    Enable := NOT gc_b_sim_on AND axisdata[2].Axis_Inbb,
    ParameterNumber := FP_S_0_0051,
    Axis := drive2,
    Value => r_motorencoder_2); // MB_ReadRealParameter

// NETWORK 17
//   axisdata[3].Axis_Inbb: A-0-0021.13 -RD- Axis is ready for power to the amplifier (bb)
//   FP_S_0_0051: Position feedback value 1
//   drive3: Real axis "Drive3" with axis number 3
FB_readmotorencoder3(
    Enable := NOT gc_b_sim_on AND axisdata[3].Axis_Inbb,
    ParameterNumber := FP_S_0_0051,
    Axis := drive3,
    Value => r_motorencoder_3); // MB_ReadRealParameter

// NETWORK 18 (disabled)
//   axisdata[4].Axis_Inbb: A-0-0021.13 -RD- Axis is ready for power to the amplifier (bb)
//   FP_S_0_0051: Position feedback value 1
//   drive4: Real axis "Drive4" with axis number 4
// FB_readmotorencoder4(
//     Enable := NOT gc_b_sim_on AND axisdata[4].Axis_Inbb,
//     ParameterNumber := FP_S_0_0051,
//     Axis := drive4,
//     Value => r_motorencoder_4); // MB_ReadRealParameter

// NETWORK 19 (disabled)
//   axisdata[5].Axis_Inbb: A-0-0021.13 -RD- Axis is ready for power to the amplifier (bb)
//   FP_S_0_0051: Position feedback value 1
//   drive5: Real axis "Drive5" with axis number 5
// FB_readmotorencoder5(
//     Enable := NOT gc_b_sim_on AND axisdata[5].Axis_Inbb,
//     ParameterNumber := FP_S_0_0051,
//     Axis := drive5,
//     Value => r_motorencoder_5); // MB_ReadRealParameter

// NETWORK 20 (disabled)
//   axisdata[6].Axis_Inbb: A-0-0021.13 -RD- Axis is ready for power to the amplifier (bb)
//   FP_S_0_0051: Position feedback value 1
//   drive6: Real axis "Drive6" with axis number 6
// FB_readmotorencoder6(
//     Enable := NOT gc_b_sim_on AND axisdata[6].Axis_Inbb,
//     ParameterNumber := FP_S_0_0051,
//     Axis := drive6,
//     Value => r_motorencoder_6); // MB_ReadRealParameter

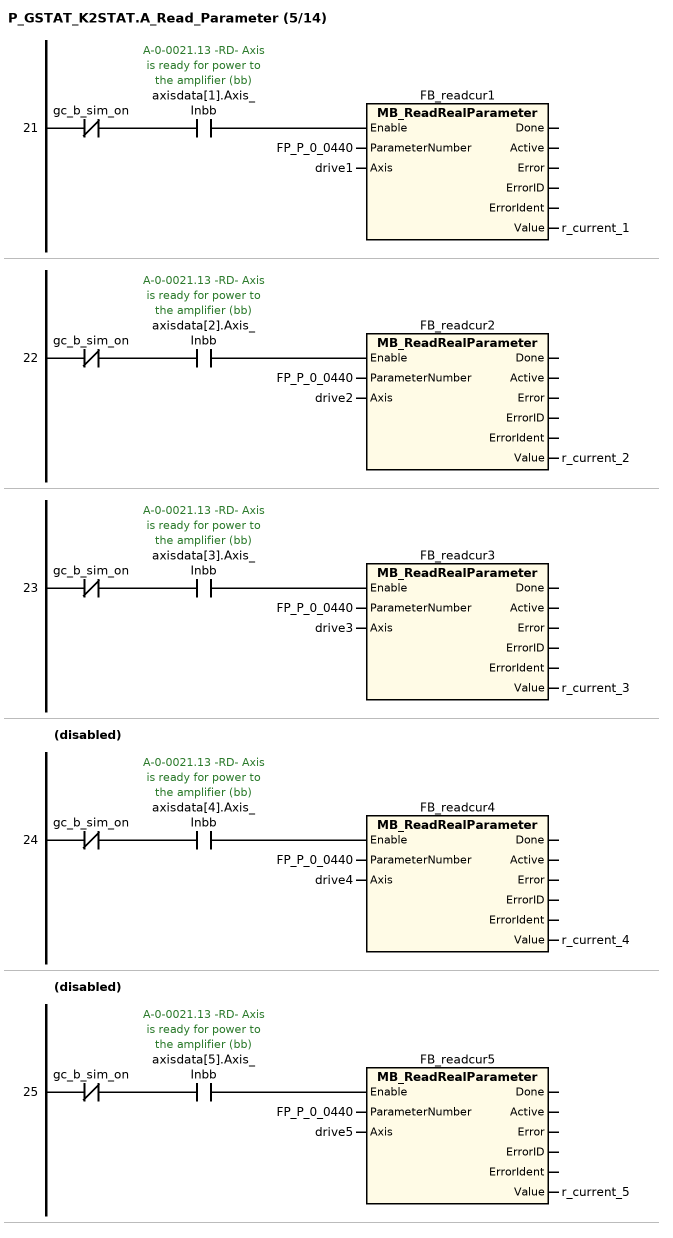
// NETWORK 21
//   FB_readcur1: With the function block "MB_ReadRealParameter" it is possible to read the current value of a parameter. The return value is REAL.
//   axisdata[1].Axis_Inbb: A-0-0021.13 -RD- Axis is ready for power to the amplifier (bb)
//   FP_P_0_0440: Actual output current value (absolute value)
//   drive1: Real axis "Drive1" with axis number 1
//   r_current_1: FP_P_0_0440,Actual output current value absolute value
FB_readcur1(
    Enable := NOT gc_b_sim_on AND axisdata[1].Axis_Inbb,
    ParameterNumber := FP_P_0_0440,
    Axis := drive1,
    Value => r_current_1); // MB_ReadRealParameter

// NETWORK 22
//   axisdata[2].Axis_Inbb: A-0-0021.13 -RD- Axis is ready for power to the amplifier (bb)
//   FP_P_0_0440: Actual output current value (absolute value)
//   drive2: Real axis "Drive2" with axis number 2
FB_readcur2(
    Enable := NOT gc_b_sim_on AND axisdata[2].Axis_Inbb,
    ParameterNumber := FP_P_0_0440,
    Axis := drive2,
    Value => r_current_2); // MB_ReadRealParameter

// NETWORK 23
//   axisdata[3].Axis_Inbb: A-0-0021.13 -RD- Axis is ready for power to the amplifier (bb)
//   FP_P_0_0440: Actual output current value (absolute value)
//   drive3: Real axis "Drive3" with axis number 3
FB_readcur3(
    Enable := NOT gc_b_sim_on AND axisdata[3].Axis_Inbb,
    ParameterNumber := FP_P_0_0440,
    Axis := drive3,
    Value => r_current_3); // MB_ReadRealParameter

// NETWORK 24 (disabled)
//   axisdata[4].Axis_Inbb: A-0-0021.13 -RD- Axis is ready for power to the amplifier (bb)
//   FP_P_0_0440: Actual output current value (absolute value)
//   drive4: Real axis "Drive4" with axis number 4
// FB_readcur4(
//     Enable := NOT gc_b_sim_on AND axisdata[4].Axis_Inbb,
//     ParameterNumber := FP_P_0_0440,
//     Axis := drive4,
//     Value => r_current_4); // MB_ReadRealParameter

// NETWORK 25 (disabled)
//   axisdata[5].Axis_Inbb: A-0-0021.13 -RD- Axis is ready for power to the amplifier (bb)
//   FP_P_0_0440: Actual output current value (absolute value)
//   drive5: Real axis "Drive5" with axis number 5
// FB_readcur5(
//     Enable := NOT gc_b_sim_on AND axisdata[5].Axis_Inbb,
//     ParameterNumber := FP_P_0_0440,
//     Axis := drive5,
//     Value => r_current_5); // MB_ReadRealParameter

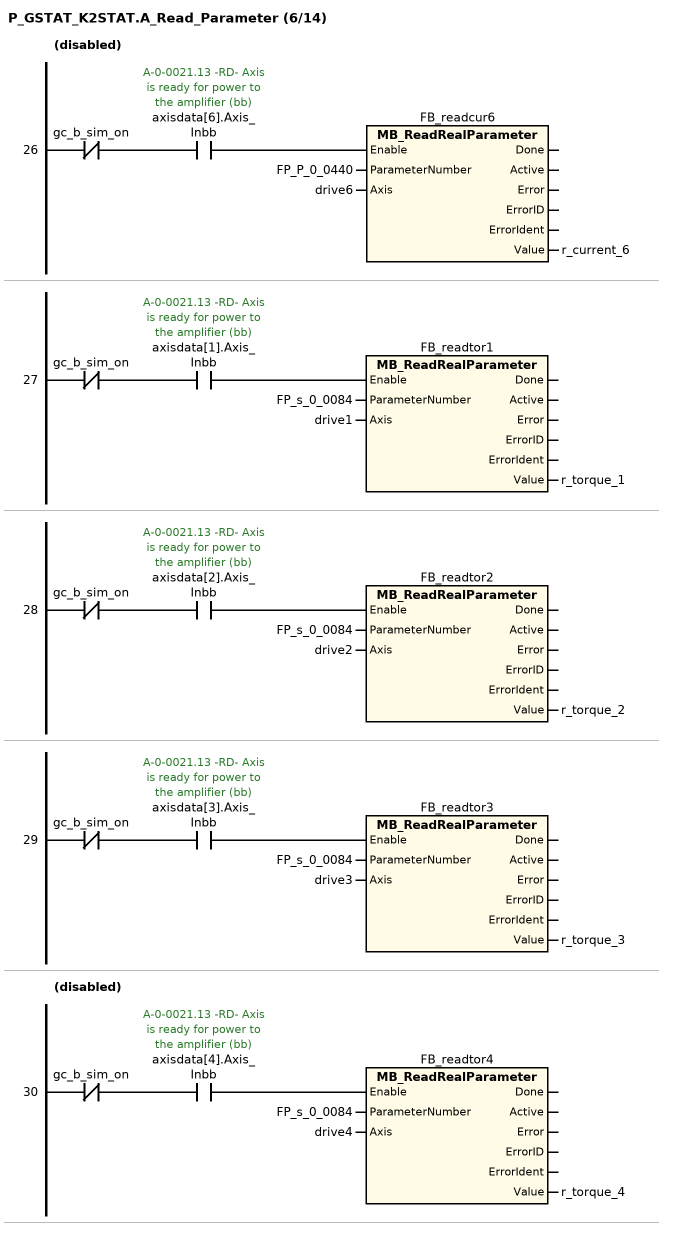
// NETWORK 26 (disabled)
//   axisdata[6].Axis_Inbb: A-0-0021.13 -RD- Axis is ready for power to the amplifier (bb)
//   FP_P_0_0440: Actual output current value (absolute value)
//   drive6: Real axis "Drive6" with axis number 6
// FB_readcur6(
//     Enable := NOT gc_b_sim_on AND axisdata[6].Axis_Inbb,
//     ParameterNumber := FP_P_0_0440,
//     Axis := drive6,
//     Value => r_current_6); // MB_ReadRealParameter

// NETWORK 27
//   axisdata[1].Axis_Inbb: A-0-0021.13 -RD- Axis is ready for power to the amplifier (bb)
//   FP_s_0_0084: Torque/force feedback value
//   drive1: Real axis "Drive1" with axis number 1
//   r_torque_1: FP_S_0_0084,Torque force feedback value
FB_readtor1(
    Enable := NOT gc_b_sim_on AND axisdata[1].Axis_Inbb,
    ParameterNumber := FP_s_0_0084,
    Axis := drive1,
    Value => r_torque_1); // MB_ReadRealParameter

// NETWORK 28
//   axisdata[2].Axis_Inbb: A-0-0021.13 -RD- Axis is ready for power to the amplifier (bb)
//   FP_s_0_0084: Torque/force feedback value
//   drive2: Real axis "Drive2" with axis number 2
FB_readtor2(
    Enable := NOT gc_b_sim_on AND axisdata[2].Axis_Inbb,
    ParameterNumber := FP_s_0_0084,
    Axis := drive2,
    Value => r_torque_2); // MB_ReadRealParameter

// NETWORK 29
//   axisdata[3].Axis_Inbb: A-0-0021.13 -RD- Axis is ready for power to the amplifier (bb)
//   FP_s_0_0084: Torque/force feedback value
//   drive3: Real axis "Drive3" with axis number 3
FB_readtor3(
    Enable := NOT gc_b_sim_on AND axisdata[3].Axis_Inbb,
    ParameterNumber := FP_s_0_0084,
    Axis := drive3,
    Value => r_torque_3); // MB_ReadRealParameter

// NETWORK 30 (disabled)
//   axisdata[4].Axis_Inbb: A-0-0021.13 -RD- Axis is ready for power to the amplifier (bb)
//   FP_s_0_0084: Torque/force feedback value
//   drive4: Real axis "Drive4" with axis number 4
// FB_readtor4(
//     Enable := NOT gc_b_sim_on AND axisdata[4].Axis_Inbb,
//     ParameterNumber := FP_s_0_0084,
//     Axis := drive4,
//     Value => r_torque_4); // MB_ReadRealParameter

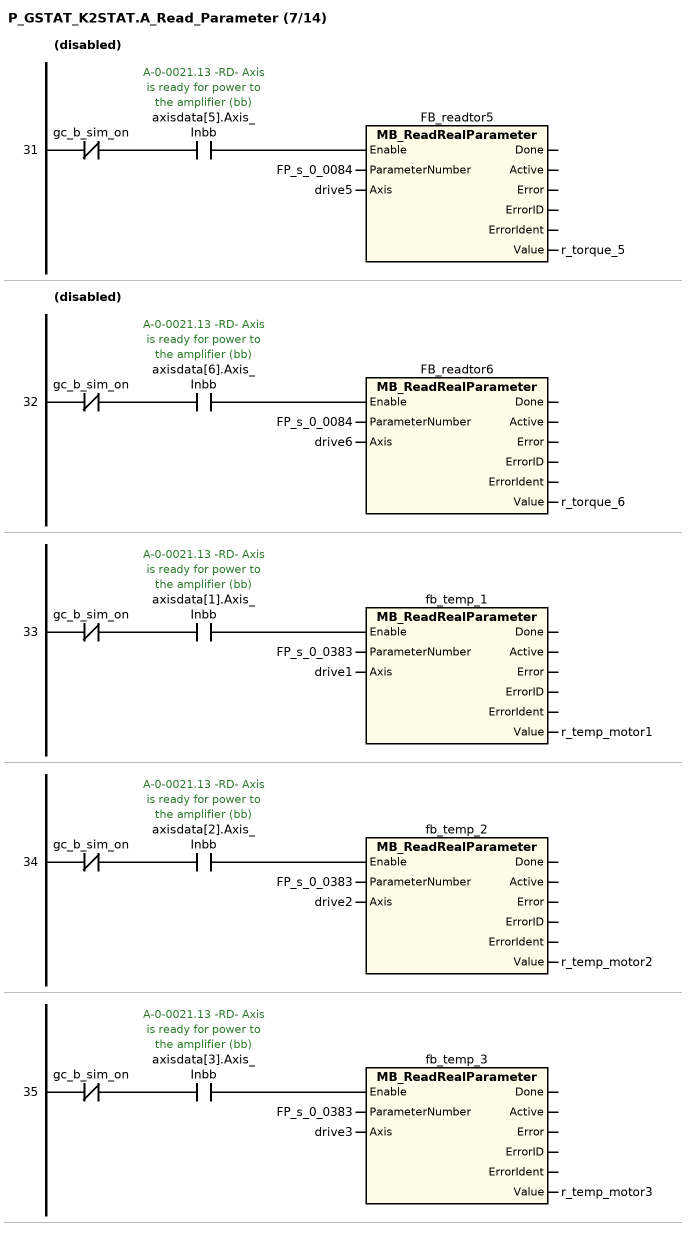
// NETWORK 31 (disabled)
//   axisdata[5].Axis_Inbb: A-0-0021.13 -RD- Axis is ready for power to the amplifier (bb)
//   FP_s_0_0084: Torque/force feedback value
//   drive5: Real axis "Drive5" with axis number 5
// FB_readtor5(
//     Enable := NOT gc_b_sim_on AND axisdata[5].Axis_Inbb,
//     ParameterNumber := FP_s_0_0084,
//     Axis := drive5,
//     Value => r_torque_5); // MB_ReadRealParameter

// NETWORK 32 (disabled)
//   axisdata[6].Axis_Inbb: A-0-0021.13 -RD- Axis is ready for power to the amplifier (bb)
//   FP_s_0_0084: Torque/force feedback value
//   drive6: Real axis "Drive6" with axis number 6
// FB_readtor6(
//     Enable := NOT gc_b_sim_on AND axisdata[6].Axis_Inbb,
//     ParameterNumber := FP_s_0_0084,
//     Axis := drive6,
//     Value => r_torque_6); // MB_ReadRealParameter

// NETWORK 33
//   axisdata[1].Axis_Inbb: A-0-0021.13 -RD- Axis is ready for power to the amplifier (bb)
//   FP_s_0_0383: Motor temperature
//   drive1: Real axis "Drive1" with axis number 1
//   r_temp_motor1: FP_S_0_0383,Motor temperature
fb_temp_1(
    Enable := NOT gc_b_sim_on AND axisdata[1].Axis_Inbb,
    ParameterNumber := FP_s_0_0383,
    Axis := drive1,
    Value => r_temp_motor1); // MB_ReadRealParameter

// NETWORK 34
//   axisdata[2].Axis_Inbb: A-0-0021.13 -RD- Axis is ready for power to the amplifier (bb)
//   FP_s_0_0383: Motor temperature
//   drive2: Real axis "Drive2" with axis number 2
fb_temp_2(
    Enable := NOT gc_b_sim_on AND axisdata[2].Axis_Inbb,
    ParameterNumber := FP_s_0_0383,
    Axis := drive2,
    Value => r_temp_motor2); // MB_ReadRealParameter

// NETWORK 35
//   axisdata[3].Axis_Inbb: A-0-0021.13 -RD- Axis is ready for power to the amplifier (bb)
//   FP_s_0_0383: Motor temperature
//   drive3: Real axis "Drive3" with axis number 3
fb_temp_3(
    Enable := NOT gc_b_sim_on AND axisdata[3].Axis_Inbb,
    ParameterNumber := FP_s_0_0383,
    Axis := drive3,
    Value => r_temp_motor3); // MB_ReadRealParameter

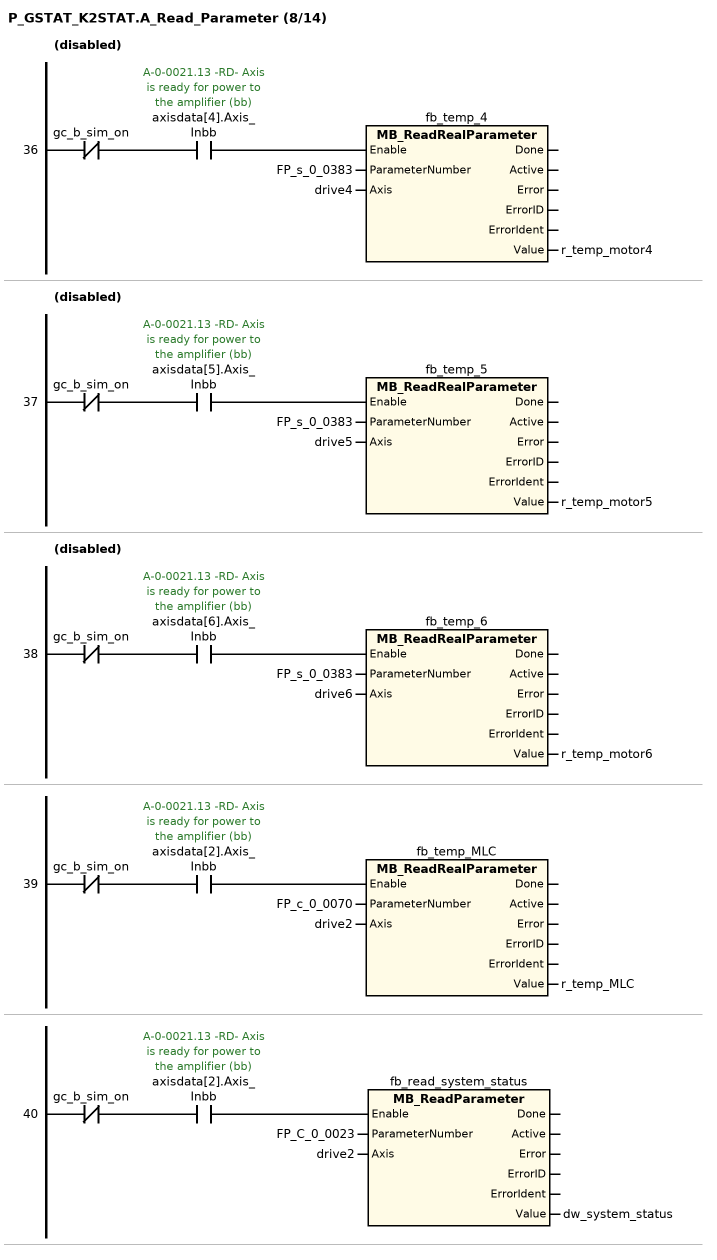
// NETWORK 36 (disabled)
//   axisdata[4].Axis_Inbb: A-0-0021.13 -RD- Axis is ready for power to the amplifier (bb)
//   FP_s_0_0383: Motor temperature
//   drive4: Real axis "Drive4" with axis number 4
// fb_temp_4(
//     Enable := NOT gc_b_sim_on AND axisdata[4].Axis_Inbb,
//     ParameterNumber := FP_s_0_0383,
//     Axis := drive4,
//     Value => r_temp_motor4); // MB_ReadRealParameter

// NETWORK 37 (disabled)
//   axisdata[5].Axis_Inbb: A-0-0021.13 -RD- Axis is ready for power to the amplifier (bb)
//   FP_s_0_0383: Motor temperature
//   drive5: Real axis "Drive5" with axis number 5
// fb_temp_5(
//     Enable := NOT gc_b_sim_on AND axisdata[5].Axis_Inbb,
//     ParameterNumber := FP_s_0_0383,
//     Axis := drive5,
//     Value => r_temp_motor5); // MB_ReadRealParameter

// NETWORK 38 (disabled)
//   axisdata[6].Axis_Inbb: A-0-0021.13 -RD- Axis is ready for power to the amplifier (bb)
//   FP_s_0_0383: Motor temperature
//   drive6: Real axis "Drive6" with axis number 6
// fb_temp_6(
//     Enable := NOT gc_b_sim_on AND axisdata[6].Axis_Inbb,
//     ParameterNumber := FP_s_0_0383,
//     Axis := drive6,
//     Value => r_temp_motor6); // MB_ReadRealParameter

// NETWORK 39
//   fb_temp_MLC: <<<<<<<<<<<<<<<<<<<<<<<<<<<<<<<<<<<<<<<add MLC temperature and operation hour(20100708)>>>>>>>>>>>>>>>>>>>>>>>>>>>>>>>>>>>>>
//   axisdata[2].Axis_Inbb: A-0-0021.13 -RD- Axis is ready for power to the amplifier (bb)
//   FP_c_0_0070: Control temperature
//   drive2: Real axis "Drive2" with axis number 2
//   r_temp_MLC: FP_c_0_0070,Control unit temperature
fb_temp_MLC(
    Enable := NOT gc_b_sim_on AND axisdata[2].Axis_Inbb,
    ParameterNumber := FP_c_0_0070,
    Axis := drive2,
    Value => r_temp_MLC); // MB_ReadRealParameter

// NETWORK 40
//   axisdata[2].Axis_Inbb: A-0-0021.13 -RD- Axis is ready for power to the amplifier (bb)
//   FP_C_0_0023: System status
//   drive2: Real axis "Drive2" with axis number 2
//   dw_system_status: FP_C_0_0023,MC system status,used for temperature warning
fb_read_system_status(
    Enable := NOT gc_b_sim_on AND axisdata[2].Axis_Inbb,
    ParameterNumber := FP_C_0_0023,
    Axis := drive2,
    Value => dw_system_status); // MB_ReadParameter

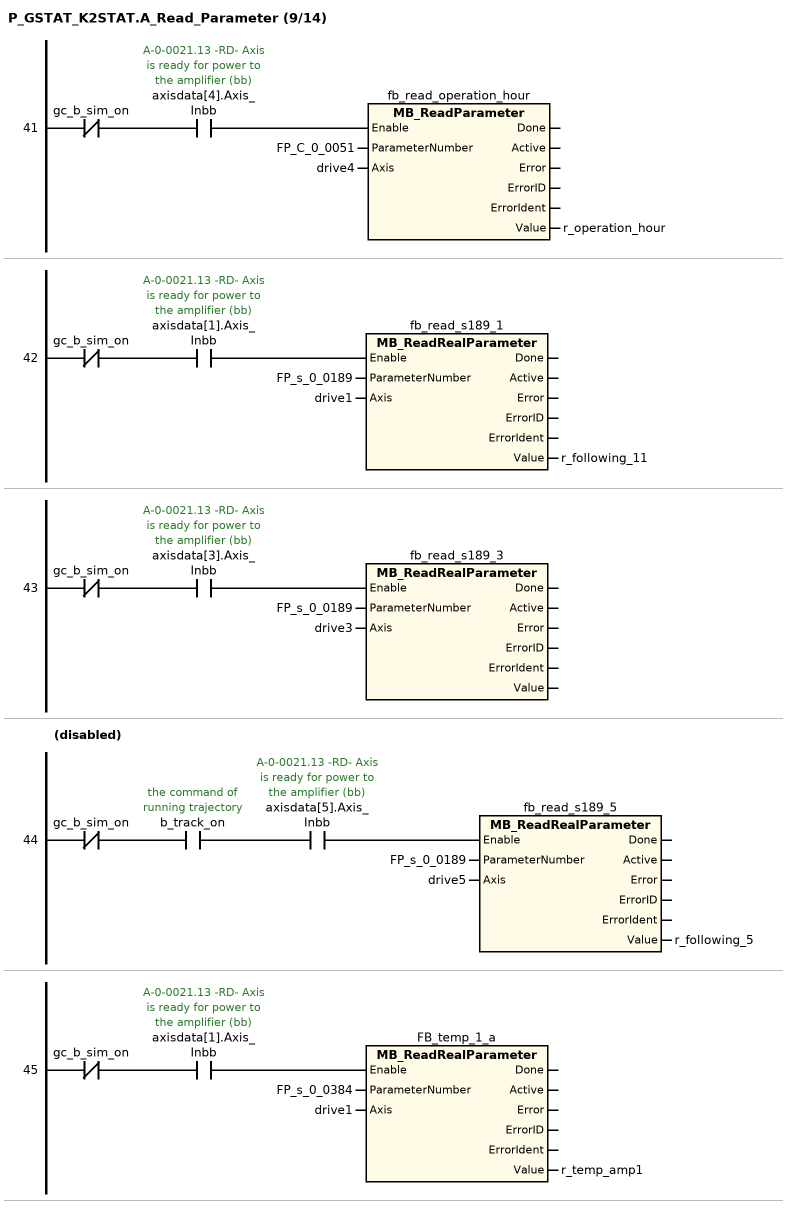
// NETWORK 41
//   axisdata[4].Axis_Inbb: A-0-0021.13 -RD- Axis is ready for power to the amplifier (bb)
//   FP_C_0_0051: Operating hour counter
//   drive4: Real axis "Drive4" with axis number 4
//   r_operation_hour: FP_C_0_0051,Operation hour counter
fb_read_operation_hour(
    Enable := NOT gc_b_sim_on AND axisdata[4].Axis_Inbb,
    ParameterNumber := FP_C_0_0051,
    Axis := drive4,
    Value => r_operation_hour); // MB_ReadParameter

// NETWORK 42
//   axisdata[1].Axis_Inbb: A-0-0021.13 -RD- Axis is ready for power to the amplifier (bb)
//   FP_s_0_0189: Following distance
//   drive1: Real axis "Drive1" with axis number 1
//   r_following_11: FP_s_0_0189,following error
fb_read_s189_1(
    Enable := NOT gc_b_sim_on AND axisdata[1].Axis_Inbb,
    ParameterNumber := FP_s_0_0189,
    Axis := drive1,
    Value => r_following_11); // MB_ReadRealParameter

// NETWORK 43
//   axisdata[3].Axis_Inbb: A-0-0021.13 -RD- Axis is ready for power to the amplifier (bb)
//   FP_s_0_0189: Following distance
//   drive3: Real axis "Drive3" with axis number 3
fb_read_s189_3(
    Enable := NOT gc_b_sim_on AND axisdata[3].Axis_Inbb,
    ParameterNumber := FP_s_0_0189,
    Axis := drive3); // MB_ReadRealParameter

// NETWORK 44 (disabled)
//   b_track_on: the command of running trajectory
//   axisdata[5].Axis_Inbb: A-0-0021.13 -RD- Axis is ready for power to the amplifier (bb)
//   FP_s_0_0189: Following distance
//   drive5: Real axis "Drive5" with axis number 5
// fb_read_s189_5(
//     Enable := NOT gc_b_sim_on AND b_track_on AND axisdata[5].Axis_Inbb,
//     ParameterNumber := FP_s_0_0189,
//     Axis := drive5,
//     Value => r_following_5); // MB_ReadRealParameter

// NETWORK 45
//   axisdata[1].Axis_Inbb: A-0-0021.13 -RD- Axis is ready for power to the amplifier (bb)
//   FP_s_0_0384: Amplifier temperature
//   drive1: Real axis "Drive1" with axis number 1
//   r_temp_amp1: FP_S_0_0384,Amplifier temperature
FB_temp_1_a(
    Enable := NOT gc_b_sim_on AND axisdata[1].Axis_Inbb,
    ParameterNumber := FP_s_0_0384,
    Axis := drive1,
    Value => r_temp_amp1); // MB_ReadRealParameter

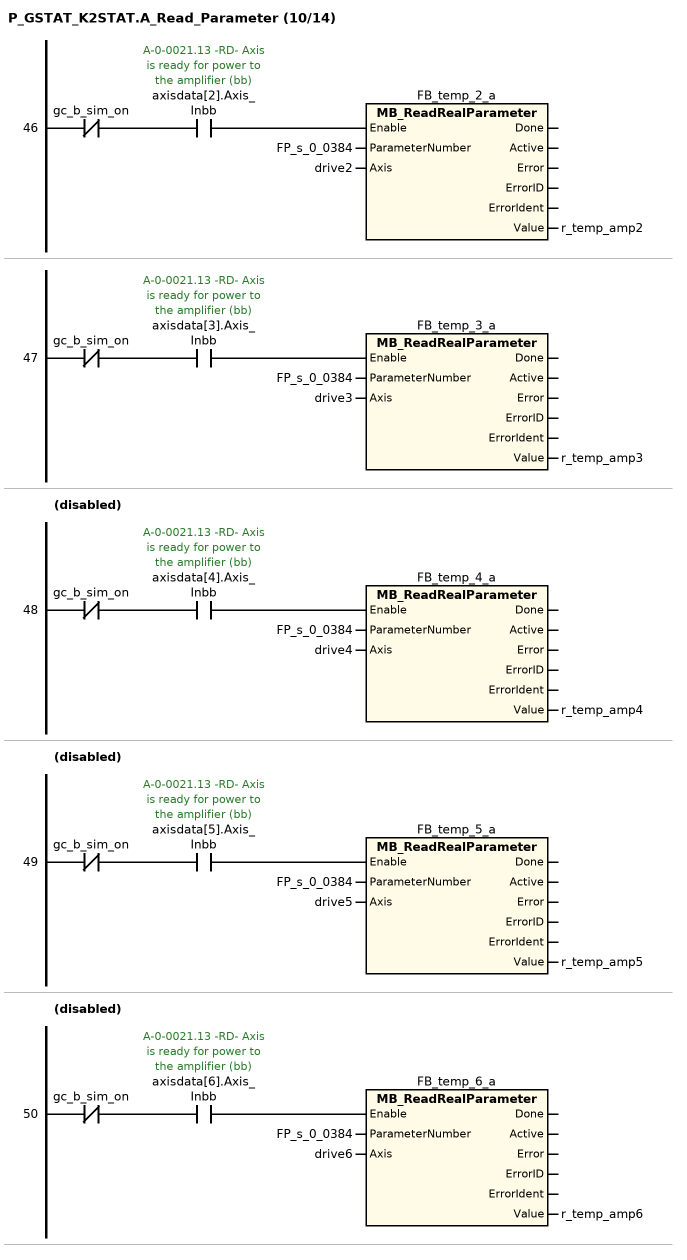
// NETWORK 46
//   axisdata[2].Axis_Inbb: A-0-0021.13 -RD- Axis is ready for power to the amplifier (bb)
//   FP_s_0_0384: Amplifier temperature
//   drive2: Real axis "Drive2" with axis number 2
FB_temp_2_a(
    Enable := NOT gc_b_sim_on AND axisdata[2].Axis_Inbb,
    ParameterNumber := FP_s_0_0384,
    Axis := drive2,
    Value => r_temp_amp2); // MB_ReadRealParameter

// NETWORK 47
//   axisdata[3].Axis_Inbb: A-0-0021.13 -RD- Axis is ready for power to the amplifier (bb)
//   FP_s_0_0384: Amplifier temperature
//   drive3: Real axis "Drive3" with axis number 3
FB_temp_3_a(
    Enable := NOT gc_b_sim_on AND axisdata[3].Axis_Inbb,
    ParameterNumber := FP_s_0_0384,
    Axis := drive3,
    Value => r_temp_amp3); // MB_ReadRealParameter

// NETWORK 48 (disabled)
//   axisdata[4].Axis_Inbb: A-0-0021.13 -RD- Axis is ready for power to the amplifier (bb)
//   FP_s_0_0384: Amplifier temperature
//   drive4: Real axis "Drive4" with axis number 4
// FB_temp_4_a(
//     Enable := NOT gc_b_sim_on AND axisdata[4].Axis_Inbb,
//     ParameterNumber := FP_s_0_0384,
//     Axis := drive4,
//     Value => r_temp_amp4); // MB_ReadRealParameter

// NETWORK 49 (disabled)
//   axisdata[5].Axis_Inbb: A-0-0021.13 -RD- Axis is ready for power to the amplifier (bb)
//   FP_s_0_0384: Amplifier temperature
//   drive5: Real axis "Drive5" with axis number 5
// FB_temp_5_a(
//     Enable := NOT gc_b_sim_on AND axisdata[5].Axis_Inbb,
//     ParameterNumber := FP_s_0_0384,
//     Axis := drive5,
//     Value => r_temp_amp5); // MB_ReadRealParameter

// NETWORK 50 (disabled)
//   axisdata[6].Axis_Inbb: A-0-0021.13 -RD- Axis is ready for power to the amplifier (bb)
//   FP_s_0_0384: Amplifier temperature
//   drive6: Real axis "Drive6" with axis number 6
// FB_temp_6_a(
//     Enable := NOT gc_b_sim_on AND axisdata[6].Axis_Inbb,
//     ParameterNumber := FP_s_0_0384,
//     Axis := drive6,
//     Value => r_temp_amp6); // MB_ReadRealParameter

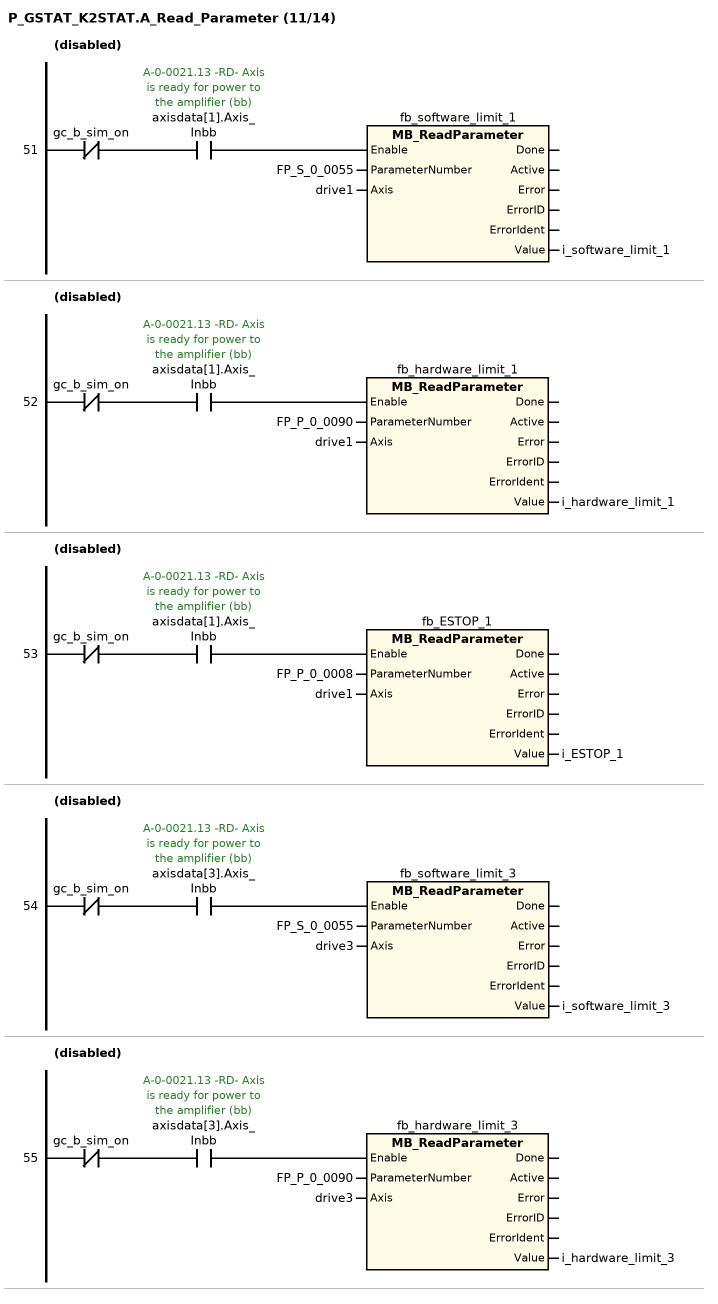
// NETWORK 51 (disabled)
//   fb_software_limit_1: test for limit check
//   axisdata[1].Axis_Inbb: A-0-0021.13 -RD- Axis is ready for power to the amplifier (bb)
//   FP_S_0_0055: Position polarities
//   drive1: Real axis "Drive1" with axis number 1
// fb_software_limit_1(
//     Enable := NOT gc_b_sim_on AND axisdata[1].Axis_Inbb,
//     ParameterNumber := FP_S_0_0055,
//     Axis := drive1,
//     Value => i_software_limit_1); // MB_ReadParameter

// NETWORK 52 (disabled)
//   axisdata[1].Axis_Inbb: A-0-0021.13 -RD- Axis is ready for power to the amplifier (bb)
//   FP_P_0_0090: Travel range limit parameter
//   drive1: Real axis "Drive1" with axis number 1
// fb_hardware_limit_1(
//     Enable := NOT gc_b_sim_on AND axisdata[1].Axis_Inbb,
//     ParameterNumber := FP_P_0_0090,
//     Axis := drive1,
//     Value => i_hardware_limit_1); // MB_ReadParameter

// NETWORK 53 (disabled)
//   axisdata[1].Axis_Inbb: A-0-0021.13 -RD- Axis is ready for power to the amplifier (bb)
//   FP_P_0_0008: Activation E-Stop function
//   drive1: Real axis "Drive1" with axis number 1
// fb_ESTOP_1(
//     Enable := NOT gc_b_sim_on AND axisdata[1].Axis_Inbb,
//     ParameterNumber := FP_P_0_0008,
//     Axis := drive1,
//     Value => i_ESTOP_1); // MB_ReadParameter

// NETWORK 54 (disabled)
//   axisdata[3].Axis_Inbb: A-0-0021.13 -RD- Axis is ready for power to the amplifier (bb)
//   FP_S_0_0055: Position polarities
//   drive3: Real axis "Drive3" with axis number 3
// fb_software_limit_3(
//     Enable := NOT gc_b_sim_on AND axisdata[3].Axis_Inbb,
//     ParameterNumber := FP_S_0_0055,
//     Axis := drive3,
//     Value => i_software_limit_3); // MB_ReadParameter

// NETWORK 55 (disabled)
//   axisdata[3].Axis_Inbb: A-0-0021.13 -RD- Axis is ready for power to the amplifier (bb)
//   FP_P_0_0090: Travel range limit parameter
//   drive3: Real axis "Drive3" with axis number 3
// fb_hardware_limit_3(
//     Enable := NOT gc_b_sim_on AND axisdata[3].Axis_Inbb,
//     ParameterNumber := FP_P_0_0090,
//     Axis := drive3,
//     Value => i_hardware_limit_3); // MB_ReadParameter

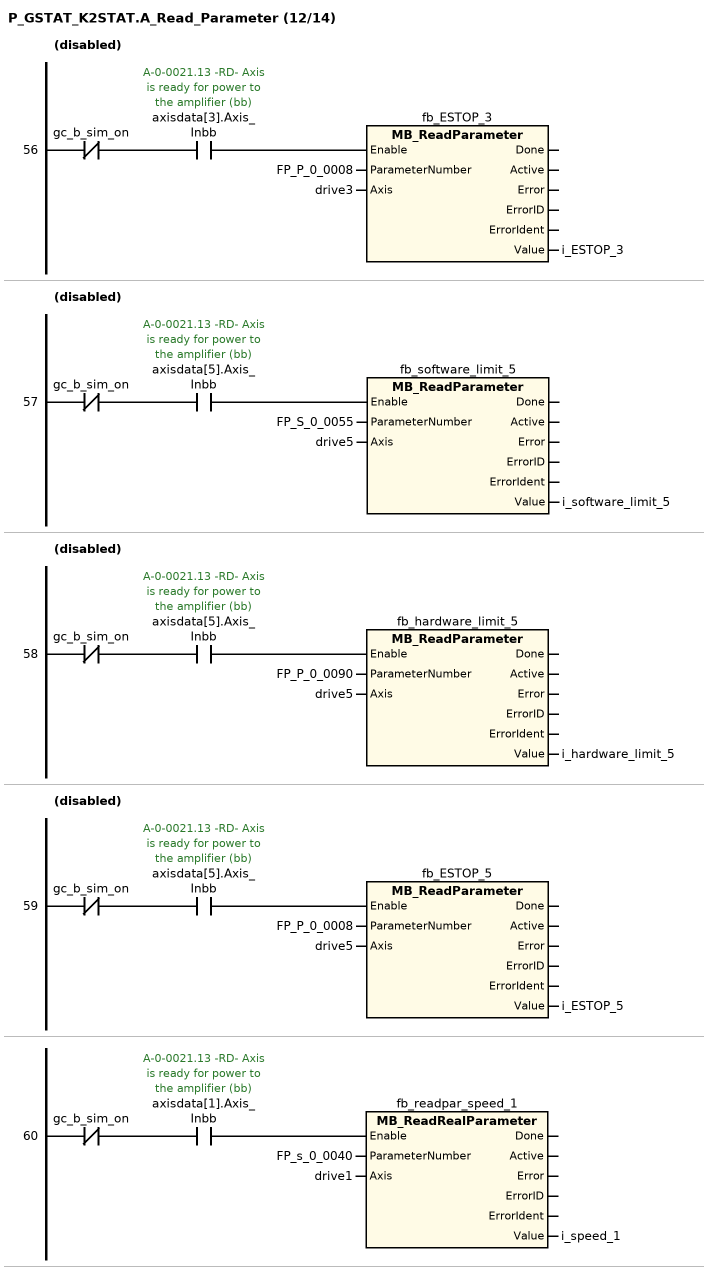
// NETWORK 56 (disabled)
//   axisdata[3].Axis_Inbb: A-0-0021.13 -RD- Axis is ready for power to the amplifier (bb)
//   FP_P_0_0008: Activation E-Stop function
//   drive3: Real axis "Drive3" with axis number 3
// fb_ESTOP_3(
//     Enable := NOT gc_b_sim_on AND axisdata[3].Axis_Inbb,
//     ParameterNumber := FP_P_0_0008,
//     Axis := drive3,
//     Value => i_ESTOP_3); // MB_ReadParameter

// NETWORK 57 (disabled)
//   axisdata[5].Axis_Inbb: A-0-0021.13 -RD- Axis is ready for power to the amplifier (bb)
//   FP_S_0_0055: Position polarities
//   drive5: Real axis "Drive5" with axis number 5
// fb_software_limit_5(
//     Enable := NOT gc_b_sim_on AND axisdata[5].Axis_Inbb,
//     ParameterNumber := FP_S_0_0055,
//     Axis := drive5,
//     Value => i_software_limit_5); // MB_ReadParameter

// NETWORK 58 (disabled)
//   axisdata[5].Axis_Inbb: A-0-0021.13 -RD- Axis is ready for power to the amplifier (bb)
//   FP_P_0_0090: Travel range limit parameter
//   drive5: Real axis "Drive5" with axis number 5
// fb_hardware_limit_5(
//     Enable := NOT gc_b_sim_on AND axisdata[5].Axis_Inbb,
//     ParameterNumber := FP_P_0_0090,
//     Axis := drive5,
//     Value => i_hardware_limit_5); // MB_ReadParameter

// NETWORK 59 (disabled)
//   axisdata[5].Axis_Inbb: A-0-0021.13 -RD- Axis is ready for power to the amplifier (bb)
//   FP_P_0_0008: Activation E-Stop function
//   drive5: Real axis "Drive5" with axis number 5
// fb_ESTOP_5(
//     Enable := NOT gc_b_sim_on AND axisdata[5].Axis_Inbb,
//     ParameterNumber := FP_P_0_0008,
//     Axis := drive5,
//     Value => i_ESTOP_5); // MB_ReadParameter

// NETWORK 60
//   axisdata[1].Axis_Inbb: A-0-0021.13 -RD- Axis is ready for power to the amplifier (bb)
//   FP_s_0_0040: Velocity feedback value
//   drive1: Real axis "Drive1" with axis number 1
//   i_speed_1: the velocity feedback value of motor1
fb_readpar_speed_1(
    Enable := NOT gc_b_sim_on AND axisdata[1].Axis_Inbb,
    ParameterNumber := FP_s_0_0040,
    Axis := drive1,
    Value => i_speed_1); // MB_ReadRealParameter

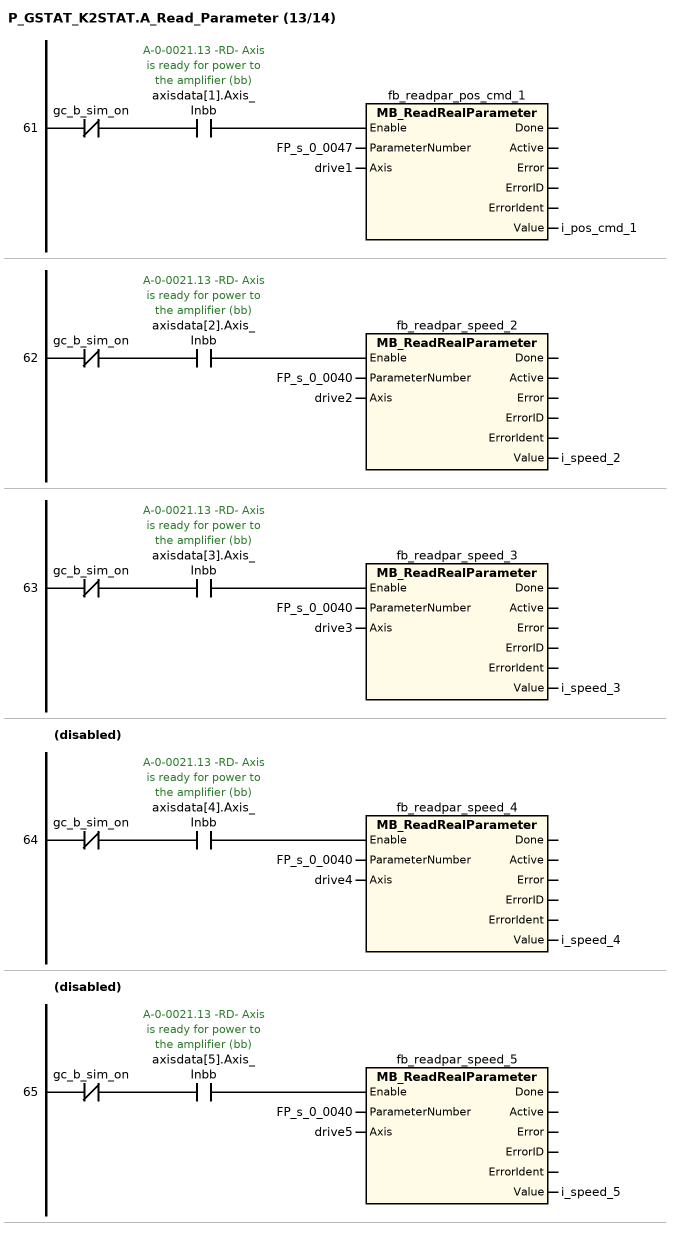
// NETWORK 61
//   axisdata[1].Axis_Inbb: A-0-0021.13 -RD- Axis is ready for power to the amplifier (bb)
//   FP_s_0_0047: Velocity feedback value
//   drive1: Real axis "Drive1" with axis number 1
//   i_pos_cmd_1: the velocity feedback value of motor1
fb_readpar_pos_cmd_1(
    Enable := NOT gc_b_sim_on AND axisdata[1].Axis_Inbb,
    ParameterNumber := FP_s_0_0047,
    Axis := drive1,
    Value => i_pos_cmd_1); // MB_ReadRealParameter

// NETWORK 62
//   axisdata[2].Axis_Inbb: A-0-0021.13 -RD- Axis is ready for power to the amplifier (bb)
//   FP_s_0_0040: Velocity feedback value
//   drive2: Real axis "Drive2" with axis number 2
//   i_speed_2: the velocity feedback value of motor1
fb_readpar_speed_2(
    Enable := NOT gc_b_sim_on AND axisdata[2].Axis_Inbb,
    ParameterNumber := FP_s_0_0040,
    Axis := drive2,
    Value => i_speed_2); // MB_ReadRealParameter

// NETWORK 63
//   axisdata[3].Axis_Inbb: A-0-0021.13 -RD- Axis is ready for power to the amplifier (bb)
//   FP_s_0_0040: Velocity feedback value
//   drive3: Real axis "Drive3" with axis number 3
//   i_speed_3: the velocity feedback value of motor3
fb_readpar_speed_3(
    Enable := NOT gc_b_sim_on AND axisdata[3].Axis_Inbb,
    ParameterNumber := FP_s_0_0040,
    Axis := drive3,
    Value => i_speed_3); // MB_ReadRealParameter

// NETWORK 64 (disabled)
//   axisdata[4].Axis_Inbb: A-0-0021.13 -RD- Axis is ready for power to the amplifier (bb)
//   FP_s_0_0040: Velocity feedback value
//   drive4: Real axis "Drive4" with axis number 4
//   i_speed_4: the velocity feedback value of motor1
// fb_readpar_speed_4(
//     Enable := NOT gc_b_sim_on AND axisdata[4].Axis_Inbb,
//     ParameterNumber := FP_s_0_0040,
//     Axis := drive4,
//     Value => i_speed_4); // MB_ReadRealParameter

// NETWORK 65 (disabled)
//   axisdata[5].Axis_Inbb: A-0-0021.13 -RD- Axis is ready for power to the amplifier (bb)
//   FP_s_0_0040: Velocity feedback value
//   drive5: Real axis "Drive5" with axis number 5
//   i_speed_5: the velocity feedback value of motor5
// fb_readpar_speed_5(
//     Enable := NOT gc_b_sim_on AND axisdata[5].Axis_Inbb,
//     ParameterNumber := FP_s_0_0040,
//     Axis := drive5,
//     Value => i_speed_5); // MB_ReadRealParameter

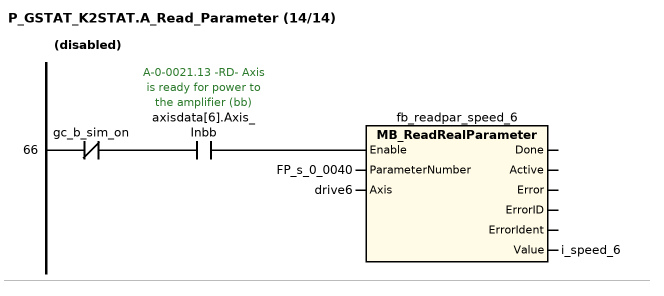
// NETWORK 66 (disabled)
//   axisdata[6].Axis_Inbb: A-0-0021.13 -RD- Axis is ready for power to the amplifier (bb)
//   FP_s_0_0040: Velocity feedback value
//   drive6: Real axis "Drive6" with axis number 6
//   i_speed_6: the velocity feedback value of motor1
// fb_readpar_speed_6(
//     Enable := NOT gc_b_sim_on AND axisdata[6].Axis_Inbb,
//     ParameterNumber := FP_s_0_0040,
//     Axis := drive6,
//     Value => i_speed_6); // MB_ReadRealParameter
END_ACTION

END_PROGRAM

// IndraMotionMlc1/Application/POUs/TCP/Message/F_reduce_to_1_bit
FUNCTION F_reduce_to_1_bit : LREAL
VAR_INPUT
	str_input: STRING(255);
END_VAR
VAR
	lr_input: LREAL;
	dint_integer: DINT;
	ui_number: UINT;
	ui_len: UINT;
	str_bit2: STRING(255);
END_VAR

ui_len:=LEN(str_input);
ui_number:=FIND(str_input,'.');
IF ui_number>0 AND ui_len-ui_number>1 THEN
	F_reduce_to_1_bit:=STRING_TO_LREAL(LEFT(str_input,ui_number+1));
	str_bit2:=MID(str_input,1,ui_number+2);
	IF STRING_TO_INT(str_bit2)>4 THEN
		F_reduce_to_1_bit:=F_reduce_to_1_bit+0.1;
	END_IF
ELSE
	F_reduce_to_1_bit:=STRING_TO_LREAL(str_input);
END_IF;

END_FUNCTION

// IndraMotionMlc1/Application/POUs/TCP/Message/F_reduce_to_4_bit
FUNCTION F_reduce_to_4_bit : LREAL
VAR_INPUT
	str_input: STRING;
END_VAR
VAR
	lr_input: LREAL;


	dint_integer: DINT;
	ui_number: UINT;
	ui_len: UINT;
	str_bit5: STRING;
END_VAR

ui_len:=LEN(str_input);
ui_number:=FIND(str_input,'.');
IF ui_number>0 AND ui_len-ui_number>4 THEN
	F_reduce_to_4_bit:=STRING_TO_LREAL(LEFT(str_input,ui_number+4));
	str_bit5:=MID(str_input,1,ui_number+5);
	IF STRING_TO_INT(str_bit5)>4 THEN
		F_reduce_to_4_bit:=F_reduce_to_4_bit+0.0001;
	END_IF
ELSE
	F_reduce_to_4_bit:=STRING_TO_LREAL(str_input);
END_IF;

END_FUNCTION

// IndraMotionMlc1/Application/POUs/OPCUA/OPCUA_Node/P_Opcua_Azimuth
{attribute linkalways}
PROGRAM P_Opcua_Azimuth
VAR
	
END_VAR

Azimuth.Status.allActive:=(axisdata[1].Axis_Power AND axisdata[2].Axis_Power);
Azimuth.Status.Active:=b_PID_in_az;
Azimuth.Status.AxisMoving:=NOT(axisdata[1].rActualVelocity_i=0);;
IF status_code1 = 'F2042' OR status_code2 = 'F2042' THEN
	azimuth.Status.encBoxOp:=1;
ELSE
	azimuth.Status.encBoxOp:=0;
END_IF
azimuth.Status.EStop:=b_in_Estop;
IF status_code1 = 'F2028' OR status_code2 = 'F2028' THEN
	azimuth.Status.Exceed:=1;
ELSE
	azimuth.Status.Exceed:=0;
END_IF
azimuth.Status.InitOk:=axisdata[1].Axis_Inbb AND axisdata[1].Axis_Inbb;
azimuth.Status.LimOverride:=0;
IF status_code1 = 'F2037' OR status_code2 = 'F2037' THEN
	azimuth.Status.posDevOk:=1;
ELSE
	azimuth.Status.posDevOk:=0;
END_IF

Azimuth.Status.Reset:=0;
Azimuth.Status.SectorSw:=b_zone_az;
IF azimuth.Status.AxisState=axisStatetype.Standby THEN
	azimuth.Status.Ready:=1;
ELSE
	azimuth.Status.Ready:=0;
END_IF
//azimuth.Status.p_Act:=pointing.Status.TotalPointCorr_Az+r_pos_az;
//azimuth.Status.p_Enc:=r_pos_az;
azimuth.Status.p_PointCorr:=pointing.Status.TotalPointCorr_Az;

IF gc_b_sim_on THEN
	azimuth.Status.p_Set:=r_write_position_az_out;
END_IF

//azimuth.Status.p_Set:=P_shape_value[1];
//azimuth.Status.p_Shape:= P_shape_value[1];
//azimuth.Status.p_Shape:=r_write_position_az_out;

azimuth.Status.p_Dev:=Azimuth.Status.p_Set-Azimuth.Status.p_Enc;
azimuth.Status.v_Act:=axisdata[1].rActualVelocity_i*6;
azimuth.Status.v_Shape:=axisdata[1].rActualVelocity_i*6;
azimuth.Status.v_SetMax:=r_vel_max_Az*6;
(***************AxisState**************)


IF (axisdata[1].Axis_Inbb AND axisdata[2].Axis_Inbb) THEN
	Azimuth.Status.AxisState:=axisstatetype.StartUp;
END_IF
IF (axisdata[1].Axis_InAb AND axisdata[2].Axis_InAb) THEN
	Azimuth.Status.AxisState:=axisstatetype.Standby;
END_IF

IF  b_stow_pin_limit_lock THEN
	Azimuth.Status.AxisState:=axisstatetype.Stowed;	
END_IF

IF  b_scc_enable_on OR b_activate_Az THEN
	azimuth.Status.AxisState:=AxisStateType.Activating;
END_IF

IF  b_scc_enable_off OR b_deactivate_Az THEN
	azimuth.Status.AxisState:=AxisStateType.Deactivating;
END_IF

IF b_PID_in_az THEN
	azimuth.Status.AxisState:=AxisStateType.Standstill;
END_IF

IF  b_track_on AND (ABS(axisdata[1].rActualVelocity_i) < (gc_r_vel_tracking_limit_Az-0.001)) THEN
	azimuth.Status.AxisState:=AxisStateType.Track;
END_IF

IF b_Estop_active OR b_interlock_active_Az THEN
	azimuth.Status.AxisState:=AxisStateType.Locked;
END_IF

IF (b_Estop_active OR b_interlock_active_Az) AND b_stow_pin_limit_lock  THEN
	azimuth.Status.AxisState:=AxisStateType.Locked_Stowed;
END_IF

IF axisdata[1].Stopping THEN
	azimuth.Status.AxisState:=AxisStateType.Stopping;
END_IF

IF (ABS(axisdata[1].rActualVelocity_i) > (gc_r_vel_tracking_limit_Az+0.001)) OR axisdata[7].DiscreteMotion THEN
	azimuth.Status.AxisState:=AxisStateType.Slew;
END_IF
(**********axis status end***********)

// Axis Statemachine attempt
(*
CASE Azimuth.Status.AxisState OF
	AxisStatetype.Activating:
       IF b_PID_in_az THEN // exit condition 
       		Azimuth.Status.AxisState:=AxisStatetype.Standstill;
       END_IF
	AxisStatetype.Deactivating:
	  IF b_power_az = False Then 
	     Azimuth.Status.AxisState:=AxisStatetype.Standby;
      End_IF
	AxisStatetype.Jog:
	  IF b_local_on AND NOT(Azimuth.Status.AxisMoving) THEN 
		 Azimuth.Status.AxisState:=AxisStateType.Standstill;
	  END_IF
	AxisStatetype.Locked:
	   IF NOT(b_interlock_active_Az) THEN
		   Azimuth.Status.AxisState:=AxisStateType.Standby;
	   END_IF
	AxisStatetype.Locked_Stowed:
	   IF NOT(b_interlock_active_Az) AND NOT(b_Estop_active) THEN
		   Azimuth.Status.AxisState:=AxisStateType.Stowed;
	   END_IF
	AxisStatetype.Slew:
         IF b_track_on AND Management.Status.OnSource THEN
           Azimuth.Status.AxisState:=AxisStateType.Track;
		 ELSIF b_stop_Az OR b_deactivate_Az OR b_Estop_active THEN
			  Azimuth.Status.AxisState:=AxisStateType.Stopping;
		 END_IF
			 
	AxisStatetype.Standby:
         IF b_enable_Az OR b_activate_Az THEN 
  			Azimuth.Status.AxisState:=AxisStateType.Activating;
		 END_IF
	AxisStatetype.Standstill:
	    IF b_local_on AND Azimuth.Status.AxisMoving THEN 
			Azimuth.Status.AxisState:=AxisStatetype.Jog;
		ELSIF b_track_on THEN 
			Azimuth.Status.AxisState:=AxisStatetype.Track;
		ELSIF b_moving_Az THEN
	        Azimuth.Status.AxisState:=AxisStatetype.Slew;
		ELSIF b_deactivate_Az THEN 
			Azimuth.Status.AxisState:=AxisStatetype.Deactivating;
		END_IF
	AxisStatetype.StartUp:
		IF (axisdata[1].Axis_InAb AND axisdata[2].Axis_InAb) THEN
			Azimuth.Status.AxisState:=axisstatetype.Standby;
        END_IF					
	AxisStatetype.Stopping:
		IF NOT(Azimuth.Status.AxisMoving) THEN
		   Azimuth.Status.AxisState:=AxisStateType.Standstill;
		END_IF
	AxisStatetype.Stowed:
		IF b_stow_pin_limit_unlock THEN
			Azimuth.Status.AxisState:=axisstatetype.Standby;
        END_IF		
	AxisStatetype.Track:
          IF NOT b_track_on THEN 
			Azimuth.Status.AxisState:=AxisStateType.Stopping;
		  ELSIF (axisdata[1].rActualVelocity_i > r_vel_tracking_limit_Az) THEN
			Azimuth.Status.AxisState:=AxisStateType.Slew;
		  ELSIF b_stop_Az OR b_deactivate_Az THEN
			  Azimuth.Status.AxisState:=AxisStateType.Stopping;
		 END_IF
	
			  
END_CASE
*)




(******ErrorStatus******)
IF axisdata[1].Axis_Error OR axisdata[2].Axis_Error THEN
	azimuth.ErrorStatus.errErrorActive:=1;
ELSE
	azimuth.ErrorStatus.errErrorActive:=0;
END_IF
azimuth.ErrorStatus.errFieldBus:=0;
azimuth.ErrorStatus.errLim2CCW:=b_limit_final_ccw_az;
azimuth.ErrorStatus.errLim2CW:=b_limit_final_cw_az;
IF status_code1 = 'E2059' OR status_code2 = 'E2059' THEN
	azimuth.ErrorStatus.errLimV_Err:=1;
ELSE
	azimuth.ErrorStatus.errLimV_Err:=0;
END_IF
azimuth.ErrorStatus.errMotComm:=(axisdata[1].Axis_NRT OR axisdata[2].Axis_NRT);
IF status_code1 = 'F2031' OR status_code2 = 'F2031' THEN
	azimuth.ErrorStatus.errMotEnc:=1;
ELSE
	azimuth.ErrorStatus.errMotEnc:=0;
END_IF
IF status_code1 = 'F2021' OR status_code2 = 'F2021' OR azimuth.ErrorStatus.errMotEnc THEN
	azimuth.ErrorStatus.errMotor:=1;
ELSE
	azimuth.ErrorStatus.errMotor:=0;
END_IF
IF azimuth.ErrorStatus.errMotor OR azimuth.ErrorStatus.errMotEnc THEN
	azimuth.ErrorStatus.errMotReady:=1;
ELSE
	azimuth.ErrorStatus.errMotReady:=0;
END_IF
azimuth.ErrorStatus.errOverride:=0;
azimuth.ErrorStatus.errV_DevExceed:=azimuth.ErrorStatus.errLimV_Err;
IF status_code1 = 'F2075' THEN
	azimuth.ErrorStatus.errP_RangeExceed:=1;
ELSE
	azimuth.ErrorStatus.errP_RangeExceed:=0;
END_IF
IF status_code1 = 'F2037' OR status_code2 = 'F2037' THEN
	azimuth.ErrorStatus.errP_DevExceed:=1;
ELSE
	azimuth.ErrorStatus.errP_DevExceed:=0;
END_IF
azimuth.ErrorStatus.errPosEnc:=azimuth.Status.encBoxOp;
azimuth.ErrorStatus.errPosEnc_Fo:=azimuth.Status.encBoxOp;
IF status_code1 = 'F2026' OR status_code2 = 'F2026' THEN
	azimuth.ErrorStatus.errPower:=1;
ELSE
	azimuth.ErrorStatus.errPower:=0;
END_IF
(***** Error status end*****)


(*******Warning state********)
azimuth.WarningStatus.waLim1CW:=b_limit_cw_az;
azimuth.WarningStatus.waLim1CCW:=b_limit_ccw_az;
IF status_code1 = 'E8029' OR status_code2 = 'E8029' THEN
	azimuth.WarningStatus.waLimSoftCW:=1;
ELSE
	azimuth.WarningStatus.waLimSoftCW:=0;
END_IF
IF status_code1 = 'E8030' OR status_code2 = 'E8030' THEN
	azimuth.WarningStatus.waLimSoftCCW:=1;
ELSE
	azimuth.WarningStatus.waLimSoftCCW:=0;
END_IF
IF status_code1 = 'E8260' OR status_code2 = 'E8260' THEN
	azimuth.WarningStatus.waMmaxExceeded:=1;
ELSE
	azimuth.WarningStatus.waMmaxExceeded:=0;
END_IF
azimuth.WarningStatus.waMotReady:=azimuth.ErrorStatus.errMotReady;
azimuth.WarningStatus.waMotWarn:=(axisdata[1].Axis_Warning OR axisdata[1].Axis_Warning);
azimuth.WarningStatus.waOverride:=0;
azimuth.WarningStatus.waParamFault:=(azimuth.WarningStatus.waMotReady OR azimuth.ErrorStatus.errMotReady);
IF status_code1 = 'E2031' OR status_code2 = 'E2031' THEN
	azimuth.WarningStatus.waPosEncWarn:=1;
ELSE
	azimuth.WarningStatus.waPosEncWarn:=0;
END_IF
azimuth.WarningStatus.waStowPinsDep:=b_stow_pin_limit_lock;
azimuth.WarningStatus.waVelLimit:=azimuth.ErrorStatus.errV_DevExceed;
(*********Warning status end***********)
(*****motor1****)
azimuth.MotorOne.ErrorCode:= STRING_TO_UINT(status_code1);
azimuth.MotorOne.mActTorq:=r_torque_1*60.5;
azimuth.MotorOne.mActVelocity:=i_speed_1;
azimuth.MotorOne.MotorTemp:=r_temp_motor1;
azimuth.MotorOne.RateOfUtil:=r_torque_1;
azimuth.MotorOne.MotorOverload:=r_torque_1;
(*****motor2****)
azimuth.MotorTwo.ErrorCode:= STRING_TO_UINT(status_code2);
azimuth.MotorTwo.mActTorq:=r_torque_2*60.5;
azimuth.MotorTwo.mActVelocity:=i_speed_2;
azimuth.MotorTwo.MotorTemp:=r_temp_motor2;
azimuth.MotorTwo.RateOfUtil:=r_torque_2;
azimuth.MotorTwo.MotorOverload:=r_torque_2;

END_PROGRAM

// IndraMotionMlc1/Application/POUs/OPCUA/OPCUA_Node/P_Opcua_Elevation
PROGRAM P_Opcua_Elevation
VAR
	
END_VAR

Elevation.Status.AllActive:=axisdata[3].Axis_Power;
Elevation.Status.Active:=axisdata[3].Axis_InSynchron;
Elevation.Status.AxisMoving:=NOT(axisdata[3].rActualVelocity_i=0);
IF status_code3 = 'F2042' OR status_code4 = 'F2042' THEN
	Elevation.Status.encBoxOp:=1;
ELSE
	Elevation.Status.encBoxOp:=0;
END_IF
Elevation.Status.EStop:=b_in_Estop;
IF status_code3 = 'F2028'THEN
	Elevation.Status.Exceed:=1;
ELSE
	Elevation.Status.Exceed:=0;
END_IF
Elevation.Status.InitOk:=axisdata[3].Axis_Inbb;
Elevation.Status.LimOverride:=0;
IF status_code3 = 'F2037' THEN
	Elevation.Status.posDevOk:=1;
ELSE
	Elevation.Status.posDevOk:=0;
END_IF

Elevation.Status.Reset:=0;
Elevation.Status.SectorSw:=b_zone_az;
IF Elevation.Status.AxisState=axisStatetype.Standby THEN
	Elevation.Status.Ready:=1;
ELSE
	Elevation.Status.Ready:=0;
END_IF
//Elevation.Status.p_Act:=pointing.Status.TotalPointCorr_El+r_pos_el;
//Elevation.Status.p_Enc:=r_pos_el;
Elevation.Status.p_PointCorr:=pointing.Status.TotalPointCorr_El;
IF gc_b_sim_on THEN
	Elevation.Status.p_Set:=r_write_position_el_out;
END_IF

//Elevation.Status.p_Set:=P_shape_value[3];
//Elevation.Status.p_Shape:= P_shape_value[3];
Elevation.Status.p_Shape:=r_write_position_el_out;
Elevation.Status.p_Dev:=Elevation.Status.p_Shape-Elevation.Status.p_Enc;
Elevation.Status.v_Act:=axisdata[3].rActualVelocity_i*6;
Elevation.Status.v_Shape:=axisdata[3].rActualVelocity_i*6;
Elevation.Status.v_SetMax:= r_vel_max_El*6;
//Elevation.Status.v_Act:=V_act_value[3];
//Elevation.Status.v_Shape:=V_shape_value[3];


(***************AxisState**************)

IF axisdata[3].Axis_Inbb  THEN
	Elevation.Status.AxisState:=axisstatetype.StartUp;
END_IF
IF axisdata[3].Axis_InAb  THEN
	Elevation.Status.AxisState:=axisstatetype.Standby;
END_IF

IF  b_stow_pin_limit_lock THEN
	Elevation.Status.AxisState:=axisstatetype.Stowed;	
END_IF

IF  b_scc_enable_on OR b_activate_El THEN
	Elevation.Status.AxisState:=AxisStateType.Activating;
END_IF

IF  b_scc_enable_off OR b_deactivate_El THEN
	Elevation.Status.AxisState:=AxisStateType.Deactivating;
END_IF

IF b_PID_in_El THEN
	Elevation.Status.AxisState:=AxisStateType.Standstill;
END_IF

IF  b_track_on AND (ABS(axisdata[3].rActualVelocity_i) < gc_r_vel_tracking_limit_El) THEN
	Elevation.Status.AxisState:=AxisStateType.Track;
END_IF

IF b_Estop_active OR b_interlock_active_El THEN
	Elevation.Status.AxisState:=AxisStateType.Locked;
END_IF

IF (b_Estop_active OR b_interlock_active_El) AND b_stow_pin_limit_lock  THEN
	Elevation.Status.AxisState:=AxisStateType.Locked_Stowed;
END_IF

IF axisdata[3].Stopping THEN
	Elevation.Status.AxisState:=AxisStateType.Stopping;
END_IF

IF (ABS(axisdata[3].rActualVelocity_i) > gc_r_vel_tracking_limit_El) OR axisdata[8].DiscreteMotion THEN
	Elevation.Status.AxisState:=AxisStateType.Slew;
END_IF
(**********axis status end***********)


(******ErrorStatus******)
IF axisdata[3].Axis_Error THEN
	Elevation.ErrorStatus.errErrorActive:=1;
ELSE
	Elevation.ErrorStatus.errErrorActive:=0;
END_IF
Elevation.ErrorStatus.errFieldBus:=0;
Elevation.ErrorStatus.errLim2CCW:=b_limit_final_ccw_el;
Elevation.ErrorStatus.errLim2CW:=b_limit_final_cw_el;
IF status_code3 = 'E2059' THEN
	Elevation.ErrorStatus.errLimV_Err:=1;
ELSE
	Elevation.ErrorStatus.errLimV_Err:=0;
END_IF
Elevation.ErrorStatus.errMotComm:=(axisdata[3].Axis_NRT OR axisdata[2].Axis_NRT);
IF status_code3 = 'F2031' THEN
	Elevation.ErrorStatus.errMotEnc:=1;
ELSE
	Elevation.ErrorStatus.errMotEnc:=0;
END_IF
IF status_code3 = 'F2021' OR Elevation.ErrorStatus.errMotEnc THEN
	Elevation.ErrorStatus.errMotor:=1;
ELSE
	Elevation.ErrorStatus.errMotor:=0;
END_IF
IF Elevation.ErrorStatus.errMotor OR Elevation.ErrorStatus.errMotEnc THEN
	Elevation.ErrorStatus.errMotReady:=1;
ELSE
	Elevation.ErrorStatus.errMotReady:=0;
END_IF
Elevation.ErrorStatus.errOverride:=0;
Elevation.ErrorStatus.errV_DevExceed:=Elevation.ErrorStatus.errLimV_Err;
IF status_code3 = 'F2075' THEN
	Elevation.ErrorStatus.errP_RangeExceed:=1;
ELSE
	Elevation.ErrorStatus.errP_RangeExceed:=0;
END_IF
IF status_code3 = 'F2037' THEN
	Elevation.ErrorStatus.errP_DevExceed:=1;
ELSE
	Elevation.ErrorStatus.errP_DevExceed:=0;
END_IF
Elevation.ErrorStatus.errPosEnc:=Elevation.Status.encBoxOp;
Elevation.ErrorStatus.errPosEnc_Fo:=Elevation.Status.encBoxOp;
IF status_code3 = 'F2026' THEN
	Elevation.ErrorStatus.errPower:=1;
ELSE
	Elevation.ErrorStatus.errPower:=0;
END_IF
(***** Error status end*****)


(*******Warning state********)
Elevation.WarningStatus.waLim1CW:=b_limit_cw_el;
Elevation.WarningStatus.waLim1CCW:=b_limit_ccw_el;
IF status_code3 = 'E8029' THEN
	Elevation.WarningStatus.waLimSoftCW:=1;
ELSE
	Elevation.WarningStatus.waLimSoftCW:=0;
END_IF
IF status_code3 = 'E8030'  THEN
	Elevation.WarningStatus.waLimSoftCCW:=1;
ELSE
	Elevation.WarningStatus.waLimSoftCCW:=0;
END_IF
IF status_code3 = 'E8260' THEN
	Elevation.WarningStatus.waMmaxExceeded:=1;
ELSE
	Elevation.WarningStatus.waMmaxExceeded:=0;
END_IF
Elevation.WarningStatus.waMotReady:=Elevation.ErrorStatus.errMotReady;
Elevation.WarningStatus.waMotWarn:=axisdata[3].Axis_Warning;
Elevation.WarningStatus.waOverride:=0;
Elevation.WarningStatus.waParamFault:=Elevation.WarningStatus.waMotReady;
IF status_code3 = 'E2031' THEN
	Elevation.WarningStatus.waPosEncWarn:=1;
ELSE
	Elevation.WarningStatus.waPosEncWarn:=0;
END_IF
//Elevation.WarningStatus.waStowPinsDep:=b_limit_lock;
Elevation.WarningStatus.waVelLimit:=Elevation.ErrorStatus.errV_DevExceed;
(*********Warning status end***********)
(*****motor1****)
Elevation.MotorOne.ErrorCode:= STRING_TO_UINT(status_code3);
Elevation.MotorOne.mActTorq:=r_torque_3*82.5;
Elevation.MotorOne.mActVelocity:=i_speed_3;
Elevation.MotorOne.MotorTemp:=r_temp_motor3;
Elevation.MotorOne.RateOfUtil:=r_torque_3;
Elevation.MotorOne.MotorOverload:=r_torque_3;
(*****motor2****)
(*Elevation.MotorTwo.ErrorCode:= STRING_TO_DINT(status_code2);
Elevation.MotorTwo.mActTorq:=r_torque_2*60.5;
Elevation.MotorTwo.mActVelocity:=i_speed_2;
Elevation.MotorTwo.MotorTemp:=r_temp_motor2;
Elevation.MotorTwo.RateOfUtil:=r_torque_2;
Elevation.MotorTwo.MotorOverload:=r_torque_2;
*)

END_PROGRAM

// IndraMotionMlc1/Application/POUs/OPCUA/OPCUA_Node/P_Opcua_FeedIndexer
PROGRAM P_Opcua_FeedIndexer
VAR
END_VAR

FeedIndexer.Status.allActive:=(axisdata[5].Axis_Power AND axisdata[6].Axis_Power);
FeedIndexer.Status.Active:=b_PID_in_FI;
FeedIndexer.Status.AxisMoving:=NOT(axisdata[5].rActualVelocity_i=0);
IF status_code4 = 'F2042' OR status_code5 = 'F2042' THEN
	FeedIndexer.Status.encBoxOp:=1;
ELSE
	FeedIndexer.Status.encBoxOp:=0;
END_IF
FeedIndexer.Status.EStop:=b_in_Estop;
IF status_code4 = 'F2028' OR status_code5 = 'F2028' THEN
	FeedIndexer.Status.Exceed:=1;
ELSE
	FeedIndexer.Status.Exceed:=0;
END_IF
FeedIndexer.Status.InitOk:=axisdata[5].Axis_Inbb AND axisdata[6].Axis_Inbb;
FeedIndexer.Status.LimOverride:=0;
IF status_code4 = 'F2037' OR status_code5 = 'F2037' THEN
	FeedIndexer.Status.posDevOk:=1;
ELSE
	FeedIndexer.Status.posDevOk:=0;
END_IF

FeedIndexer.Status.Reset:=0;
//FeedIndexer.SectorSw:=b_zone_FI;
IF FeedIndexer.Status.AxisState=axisStatetype.Standby THEN
	FeedIndexer.Status.Ready:=1;
ELSE
	FeedIndexer.Status.Ready:=0;
END_IF
FeedIndexer.Status.p_Act:=r_pos_FI; 
FeedIndexer.Status.p_Enc:=r_pos_FI;
FeedIndexer.Status.p_PointCorr:=0;


//FeedIndexer.Status.p_Set:=r_write_position_fi_out;
//FeedIndexer.Status.p_Shape:= P_shape_value[4];
//FeedIndexer.Status.p_Set:=r_write_position_fi_out;
FeedIndexer.Status.p_Shape:=r_write_position_fi_out;;
FeedIndexer.Status.p_Dev:=FeedIndexer.Status.p_Set-FeedIndexer.Status.p_Enc;
//FeedIndexer.Status.v_Act:=V_act_value[4];
//FeedIndexer.Status.v_Shape:=V_shape_value[4];
FeedIndexer.Status.v_Act:=axisdata[9].rActualVelocity_i*6;
FeedIndexer.Status.v_Shape:=axisdata[9].rActualVelocity_i*6;
FeedIndexer.Status.v_SetMax:=r_vel_max_Fi*6;

	


(***************AxisState**************)
IF (axisdata[4].Axis_Inbb AND axisdata[5].Axis_Inbb) THEN
	FeedIndexer.Status.AxisState:=AxisStateType.StartUp;
END_IF
IF (axisdata[4].Axis_InAb AND axisdata[5].Axis_InAb) THEN
	FeedIndexer.Status.AxisState:=AxisStateType.Standby;
END_IF

IF  b_scc_enable_on OR b_activate_FI THEN
	FeedIndexer.Status.AxisState:=AxisStateType.Activating;
END_IF

IF  b_scc_enable_off OR b_deactivate_FI THEN
	FeedIndexer.Status.AxisState:=AxisStateType.Deactivating;
END_IF

IF b_PID_in_FI THEN
	FeedIndexer.Status.AxisState:=AxisStateType.Standstill;
END_IF


(*IF  b_track_on  THEN
	FeedIndexer.Status.AxisState:=AxisStateType.Track;
END_IF *)

IF b_Estop_active and b_interlock_active_Fi THEN
	FeedIndexer.Status.AxisState:=AxisStateType.Locked;
END_IF
IF axisdata[9].Stopping  THEN
	FeedIndexer.Status.AxisState:=AxisStateType.Stopping;
END_IF

IF ABS(axisdata[9].rActualVelocity_i) > gc_r_vel_tracking_limit_Fi THEN
	FeedIndexer.Status.AxisState:=AxisStateType.Slew;
END_IF
(**********axis status end***********)


(******ErrorStatus******)
IF axisdata[4].Axis_Error OR axisdata[5].Axis_Error THEN
	FeedIndexer.ErrorStatus.errErrorActive:=1;
ELSE
	FeedIndexer.ErrorStatus.errErrorActive:=0;
END_IF
FeedIndexer.ErrorStatus.errFieldBus:=0;
FeedIndexer.ErrorStatus.errLim2CCW:=b_limit_final_ccw_FI;
FeedIndexer.ErrorStatus.errLim2CW:=b_limit_final_cw_FI;
IF status_code4 = 'E2059' OR status_code5 = 'E2059' THEN
	FeedIndexer.ErrorStatus.errLimV_Err:=1;
ELSE
	FeedIndexer.ErrorStatus.errLimV_Err:=0;
END_IF
FeedIndexer.ErrorStatus.errMotComm:=(axisdata[5].Axis_NRT OR axisdata[6].Axis_NRT);
IF status_code4 = 'F2031' OR status_code5 = 'F2031' THEN
	FeedIndexer.ErrorStatus.errMotEnc:=1;
ELSE
	FeedIndexer.ErrorStatus.errMotEnc:=0;
END_IF
IF status_code4 = 'F2021' OR status_code5 = 'F2021' OR FeedIndexer.ErrorStatus.errMotEnc THEN
	FeedIndexer.ErrorStatus.errMotor:=1;
ELSE
	FeedIndexer.ErrorStatus.errMotor:=0;
END_IF
IF FeedIndexer.ErrorStatus.errMotor OR FeedIndexer.ErrorStatus.errMotEnc THEN
	FeedIndexer.ErrorStatus.errMotReady:=1;
ELSE
	FeedIndexer.ErrorStatus.errMotReady:=0;
END_IF
FeedIndexer.ErrorStatus.errOverride:=0;
FeedIndexer.ErrorStatus.errV_DevExceed:=FeedIndexer.ErrorStatus.errLimV_Err;
IF status_code4 = 'F2075' THEN
	FeedIndexer.ErrorStatus.errP_RangeExceed:=1;
ELSE
	FeedIndexer.ErrorStatus.errP_RangeExceed:=0;
END_IF
IF status_code4 = 'F2037' OR status_code5 = 'F2037' THEN
	FeedIndexer.ErrorStatus.errP_DevExceed:=1;
ELSE
	FeedIndexer.ErrorStatus.errP_DevExceed:=0;
END_IF
FeedIndexer.ErrorStatus.errPosEnc:=FeedIndexer.Status.encBoxOp;
FeedIndexer.ErrorStatus.errPosEnc_Fo:=FeedIndexer.Status.encBoxOp;
IF status_code4 = 'F2026' OR status_code5 = 'F2026' THEN
	FeedIndexer.ErrorStatus.errPower:=1;
ELSE
	FeedIndexer.ErrorStatus.errPower:=0;
END_IF
(***** Error status end*****)


(*******Warning state********)
FeedIndexer.WarningStatus.waLim1CW:=b_limit_cw_FI;
FeedIndexer.WarningStatus.waLim1CCW:=b_limit_ccw_FI;
IF status_code4 = 'E8029' OR status_code5 = 'E8029' THEN
	FeedIndexer.WarningStatus.waLimSoftCW:=1;
ELSE
	FeedIndexer.WarningStatus.waLimSoftCW:=0;
END_IF
IF status_code4 = 'E8030' OR status_code5 = 'E8030' THEN
	FeedIndexer.WarningStatus.waLimSoftCCW:=1;
ELSE
	FeedIndexer.WarningStatus.waLimSoftCCW:=0;
END_IF
IF status_code4 = 'E8260' OR status_code5 = 'E8260' THEN
	FeedIndexer.WarningStatus.waMmaxExceeded:=1;
ELSE
	FeedIndexer.WarningStatus.waMmaxExceeded:=0;
END_IF
FeedIndexer.WarningStatus.waMotReady:=FeedIndexer.ErrorStatus.errMotReady;
FeedIndexer.WarningStatus.waMotWarn:=(axisdata[4].Axis_Warning OR axisdata[4].Axis_Warning);
FeedIndexer.WarningStatus.waOverride:=0;
FeedIndexer.WarningStatus.waParamFault:=(FeedIndexer.WarningStatus.waMotReady OR FeedIndexer.ErrorStatus.errMotReady);
IF status_code4 = 'E2031' OR status_code5 = 'E2031' THEN
	FeedIndexer.WarningStatus.waPosEncWarn:=1;
ELSE
	FeedIndexer.WarningStatus.waPosEncWarn:=0;
END_IF
FeedIndexer.WarningStatus.waStowPinsDep:=FALSE;
FeedIndexer.WarningStatus.waVelLimit:=FeedIndexer.ErrorStatus.errV_DevExceed;
(*********Warning status end***********)
(*****motor1****)
FeedIndexer.MotorOne.ErrorCode:= STRING_TO_UINT(status_code4);
FeedIndexer.MotorOne.mActTorq:=r_torque_4*7.1;
FeedIndexer.MotorOne.mActVelocity:=i_speed_4;
FeedIndexer.MotorOne.MotorTemp:=r_temp_motor4;
FeedIndexer.MotorOne.RateOfUtil:=r_torque_4;
FeedIndexer.MotorOne.MotorOverload:=r_torque_4;
(*****motor2****)
FeedIndexer.MotorTwo.ErrorCode:= STRING_TO_UINT(status_code5);
FeedIndexer.MotorTwo.mActTorq:=r_torque_5*7.1;
FeedIndexer.MotorTwo.mActVelocity:=i_speed_5;
FeedIndexer.MotorTwo.MotorTemp:=r_temp_motor5;
FeedIndexer.MotorTwo.RateOfUtil:=r_torque_5;
FeedIndexer.MotorTwo.MotorOverload:=r_torque_5;

END_PROGRAM

// IndraMotionMlc1/Application/POUs/OPCUA/OPCUA_Node/P_Opcua_Safety
PROGRAM P_Opcua_Safety
VAR
	b_final_limit_active:BOOL;
	fb_move_stow_Az: MC_MoveAbsolute;
	fb_move_stow_El: MC_MoveAbsolute;
	fb_ton_stow: TON;
	fb_self_reset_stow: R_Trig;
	fb_ton_self_reset_stow: TON;
	fb_rtrig_off_stow:R_Trig;
	fb_rtrig_lock_stow: R_Trig;
	fb_rtrig_reset_deploy: R_Trig;
	fb_rtrig_reset_retract: R_Trig;
	fb_rtrig_estop: R_TRIG;
	fb_rtrig_interlock_Az: R_TRIG;
	fb_rtrig_interlock_El: R_TRIG;
	fb_rtrig_interlock_Fi: R_TRIG;
	
	fb_ton_sim_stow: TON;
	_retract: TON;
	fb_ton_sim_retract: TON;
	fb_ton_sim_deploy: TON;
	fb_rtrig_sim_retract: R_TRIG;
	fb_rtrig_sim_deploy: R_TRIG;
	fb_rtrig_stow_deactivate: R_TRIG;
	fb_rtrig_stow_pulse: R_TRIG;
	_test: BOOL;
	b_stow_SIP: BOOL;
	rtrig_Estop_Az: R_TRIG;
	fb_Estop_Az: MC_Stop;
	rtrig_Estop_El: R_TRIG;
	fb_Estop_El: MC_Stop;
	rtrig_Estop_Fi: R_TRIG;
	fb_Estop_Fi: MC_Stop;
	MC_MoveRelative_0: MC_MoveRelative;
	MC_MoveRelative_1: MC_MoveRelative;
	R_TRIG_0: R_TRIG;
	TON_0: TON;
	b_stow_wait: BOOL;
	TON_1: TON;
	b_stow_run: BOOL;
	R_TRIG_1: R_TRIG;
	F_TRIG_0: F_TRIG;
	F_TRIG_1: F_TRIG;
	F_TRIG_2: F_TRIG;
	F_TRIG_3: F_TRIG;
	F_TRIG_4: F_TRIG;
END_VAR
VAR // added by the converter: edge detectors and wires of the graphical bodies
    _w1, _w2, _w3, _w4, _w5 : BOOL;
END_VAR

safety();
(*IF b_HHP_Estop OR b_Turnhead_Estop OR b_DS_Estop OR b_FI_Estop OR b_Turnhead_Hatch OR b_AZ_Hatch OR (NOT(b_stow_pin_limit_unlock)) THEN
	b_in_interlock:=1;
ELSE
	b_in_interlock:=0;
END_IF*)

(*IF b_in_interlock OR b_DSDoor_Estop OR b_PSCDoor_Estop OR b_DriveCabinetDoor_Estop OR b_EMISCDoor_Estop THEN // b_in_interlock true will cause an EStop. Whereas it should only cause an interlock. 
	b_in_Estop:=1;
ELSE
	b_in_Estop:=0;
END_IF*)
safety.Status.AutoStowActive:=0;
safety.Status.Axes_InitFault:=NOT(Azimuth.Status.InitOk AND Elevation.Status.InitOk AND FeedIndexer.Status.InitOk);
safety.Status.EStopFi:=b_FI_Estop;
safety.Status.EStopHHP:=b_HHP_Estop;
safety.Status.EStopPED:=b_DS_Estop;
safety.Status.EStopTurnhead:=b_Turnhead_Estop;
safety.Status.HatchTurnheadRoof:=b_Turnhead_Hatch;
safety.Status.HatchAzBearing:=b_AZ_Hatch;
//safety.InterlockAck
safety.Status.Lim2_CCW_Az:=b_limit_final_ccw_az;
safety.Status.Lim2_CCW_Fi:=b_limit_final_ccw_Fi;
safety.Status.Lim2_CW_Az:=b_limit_final_cw_az;
safety.Status.Lim2_CW_Fi:=b_limit_final_cw_Fi;
safety.Status.Lim2_Dn_El:=b_limit_final_ccw_el;
safety.Status.Lim2_Up_El:=b_limit_final_cw_el;
b_final_limit_active:=(safety.Status.Lim2_CCW_Az OR safety.Status.Lim2_CW_Az OR safety.Status.Lim2_Dn_El OR safety.Status.Lim2_Up_El OR safety.Status.Lim2_CCW_Fi OR safety.Status.Lim2_CW_Fi); 

(* Still to be wired in *)
safety.Status.SafetyLockout_Az:=b_Lock_Out_Az;
safety.Status.SafetyLockout_El:=b_Lock_Out_El;
safety.Status.SafetyLockout_Fi:=b_Lock_Out_Fi;

IF safety.Status.Axes_InitFault THEN
	safety.Status.SafetyState:=SafetyStatetype.Stopped;
ELSIF b_in_interlock OR b_in_Estop OR b_final_limit_active THEN
	safety.Status.SafetyState:=SafetyStatetype.Error;
ELSE
	safety.Status.SafetyState:=SafetyStatetype.Running;	
END_IF
safety.Status.STO_Az:=b_in_interlock;
safety.Status.STO_El:=b_in_interlock;
safety.Status.STO_Fi:=b_in_interlock;

IF b_stow_pin_deploy AND NOT(b_stow_pin_limit_lock) THEN
	safety.Status.StowPinStatus:=StowPinStatustype.Deploying;
ELSIF b_stow_pin_limit_lock THEN
	safety.Status.StowPinStatus:=StowPinStatustype.Deployed;
ELSIF b_stow_pin_retract AND NOT(b_stow_pin_limit_unlock) THEN
	safety.Status.StowPinStatus:=StowPinStatustype.Retracting;
ELSIF b_stow_pin_limit_unlock THEN
	safety.Status.StowPinStatus:=StowPinStatustype.Retracted;
END_IF

IF (Azimuth.Status.p_Enc >= Azimuth.Status.StowPos_Minus AND Azimuth.Status.p_Enc <= Azimuth.Status.StowPos_Plus) THEN
	b_stow_lock_allow:=1;
ELSE 
	b_stow_lock_allow:=0;
END_IF

(*
IF b_in_interlock AND b_in_Estop THEN 
	Safety.Status.InterlockClearable:=0;
ELSE
	Safety.Status.InterlockClearable:=1;	
END_IF *)

// Run Ladder Logic
P_Opcua_Safety.A_STOW();
P_Opcua_Safety.A_Interlock_Estop();

ACTION A_STOW:
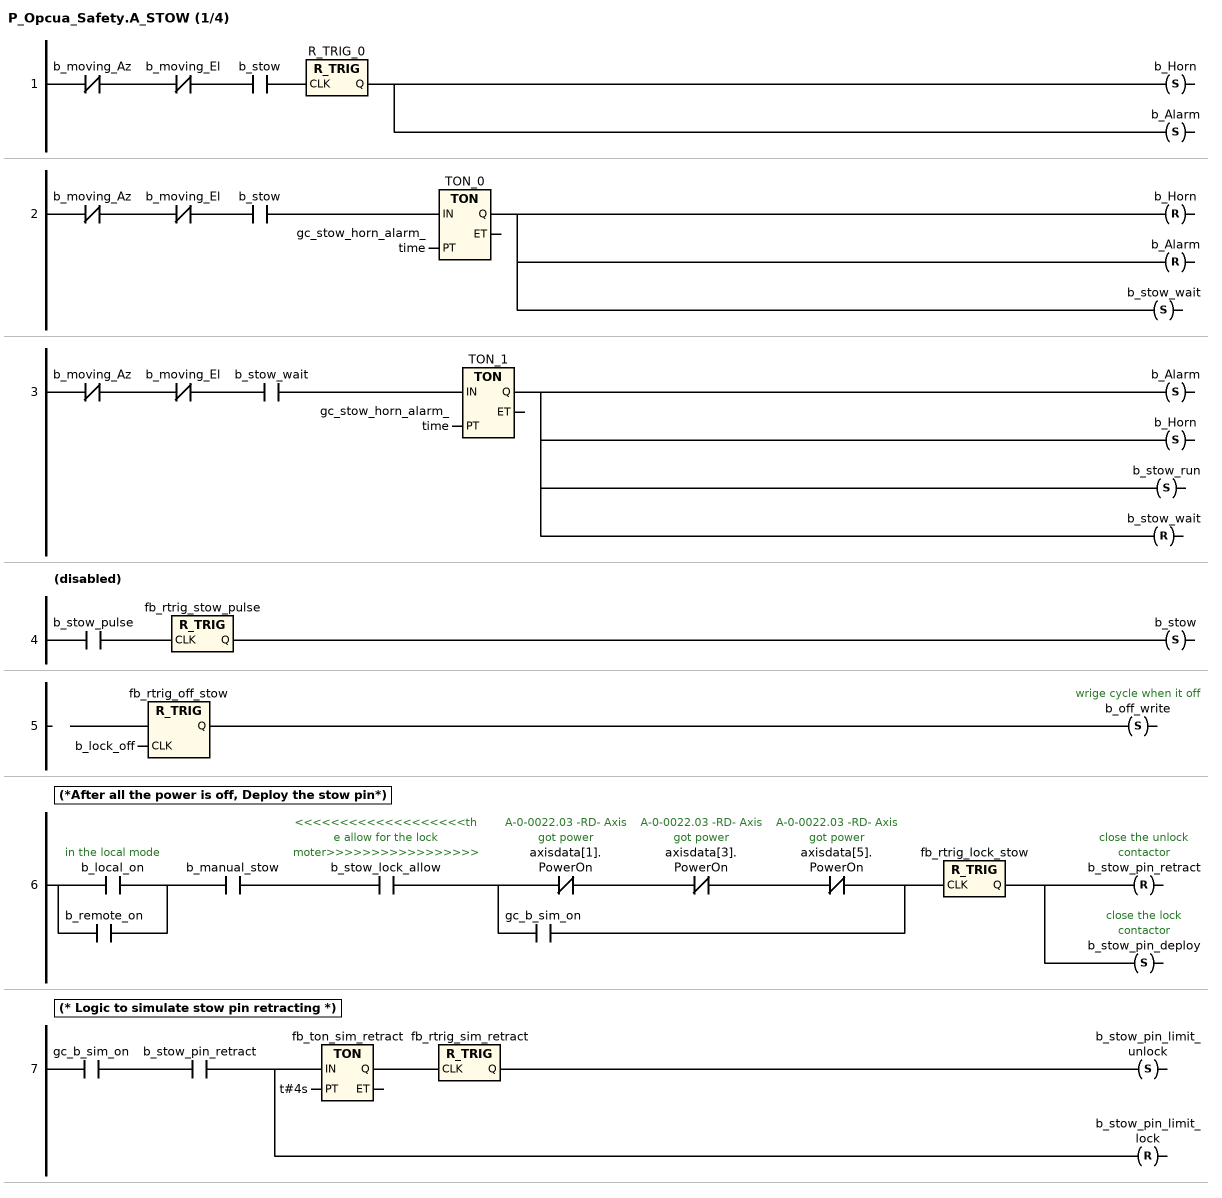
// NETWORK 1
R_TRIG_0(CLK := NOT b_moving_Az AND NOT b_moving_El AND b_stow); // R_TRIG
b_Horn S= R_TRIG_0.Q;
b_Alarm S= R_TRIG_0.Q;

// NETWORK 2
TON_0(IN := NOT b_moving_Az AND NOT b_moving_El AND b_stow, PT := gc_stow_horn_alarm_time); // TON
b_Horn R= TON_0.Q;
b_Alarm R= TON_0.Q;
b_stow_wait S= TON_0.Q;

// NETWORK 3
TON_1(IN := NOT b_moving_Az AND NOT b_moving_El AND b_stow_wait, PT := gc_stow_horn_alarm_time); // TON
b_Alarm S= TON_1.Q;
b_Horn S= TON_1.Q;
b_stow_run S= TON_1.Q;
b_stow_wait R= TON_1.Q;

// NETWORK 4 (disabled)
//   fb_rtrig_stow_pulse: the definition of rise trigger,The function block R_TRIG detects a rising edge.
// fb_rtrig_stow_pulse(CLK := b_stow_pulse); // R_TRIG
// b_stow S= fb_rtrig_stow_pulse.Q;

// NETWORK 5
//   b_lock_off: power off after arriving at the stow position
//   b_off_write: wrige cycle when it off
fb_rtrig_off_stow(CLK := b_lock_off); // R_TRIG
b_off_write S= fb_rtrig_off_stow.Q;

// NETWORK 6
//   fb_rtrig_lock_stow: the definition of rise trigger,The function block R_TRIG detects a rising edge.
//   b_local_on: in the local mode
//   b_stow_lock_allow: <<<<<<<<<<<<<<<<<<<the allow for the lock moter>>>>>>>>>>>>>>>>>
//   axisdata[1].PowerOn: A-0-0022.03 -RD- Axis got power
//   axisdata[3].PowerOn: A-0-0022.03 -RD- Axis got power
//   axisdata[5].PowerOn: A-0-0022.03 -RD- Axis got power
//   b_stow_pin_retract: close the unlock contactor
//   b_stow_pin_deploy: close the lock contactor
// label: (*After all the power is off, Deploy the stow pin*)
fb_rtrig_lock_stow(CLK := (b_local_on OR b_remote_on) AND b_manual_stow AND b_stow_lock_allow AND (NOT axisdata[1].PowerOn AND NOT axisdata[3].PowerOn AND NOT axisdata[5].PowerOn OR gc_b_sim_on)); // R_TRIG
b_stow_pin_retract R= fb_rtrig_lock_stow.Q;
b_stow_pin_deploy S= fb_rtrig_lock_stow.Q;

// NETWORK 7
//   fb_rtrig_sim_retract: the definition of rise trigger,The function block R_TRIG detects a rising edge.
//   fb_ton_sim_retract: The function block Timer On Delay implements a turn-on delay
// label: (* Logic to simulate stow pin retracting *)
_w1 := gc_b_sim_on AND b_stow_pin_retract;
fb_ton_sim_retract(IN := _w1, PT := t#4s); // TON
fb_rtrig_sim_retract(CLK := fb_ton_sim_retract.Q); // R_TRIG
b_stow_pin_limit_unlock S= fb_rtrig_sim_retract.Q;
b_stow_pin_limit_lock R= _w1;

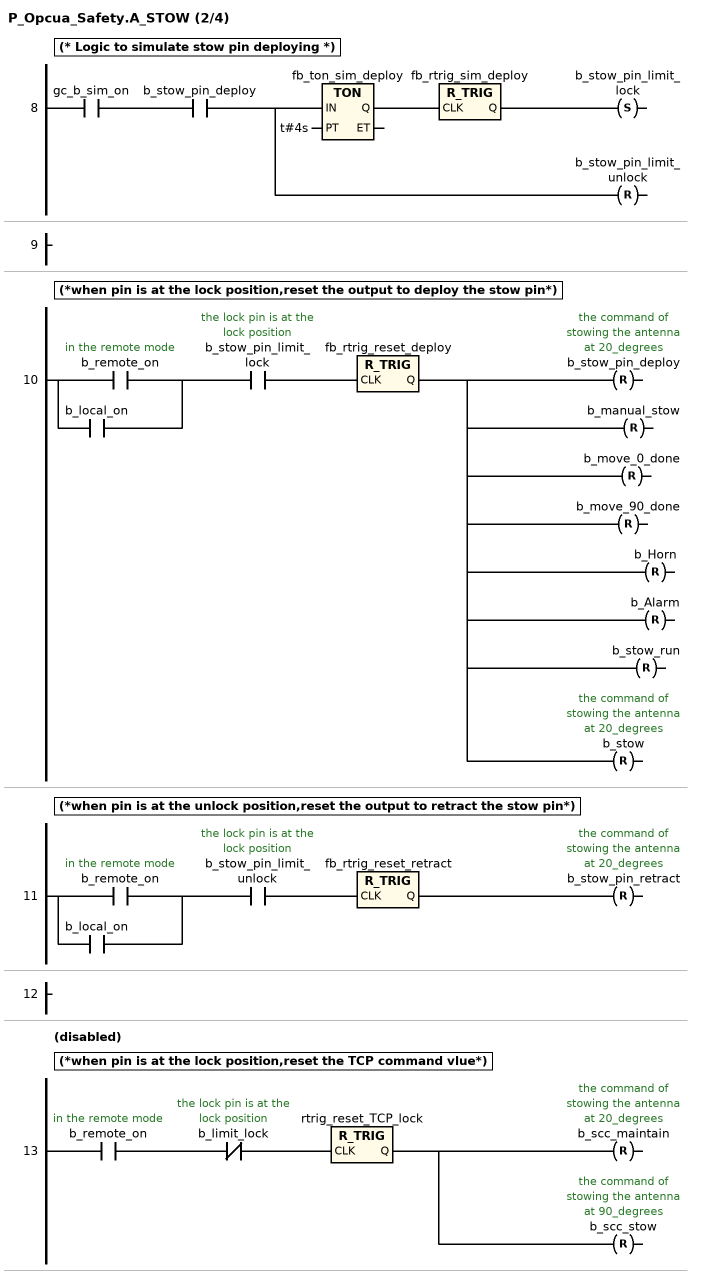
// NETWORK 8
//   fb_rtrig_sim_deploy: the definition of rise trigger,The function block R_TRIG detects a rising edge.
//   fb_ton_sim_deploy: The function block Timer On Delay implements a turn-on delay
// label: (* Logic to simulate stow pin deploying *)
_w2 := gc_b_sim_on AND b_stow_pin_deploy;
fb_ton_sim_deploy(IN := _w2, PT := t#4s); // TON
fb_rtrig_sim_deploy(CLK := fb_ton_sim_deploy.Q); // R_TRIG
b_stow_pin_limit_lock S= fb_rtrig_sim_deploy.Q;
b_stow_pin_limit_unlock R= _w2;

// NETWORK 9

// NETWORK 10
//   b_remote_on: in the remote mode
//   b_stow_pin_limit_lock: the lock pin is at the lock position
//   b_stow_pin_deploy: the command of stowing the antenna at 20_degrees
//   b_stow: the command of stowing the antenna at 20_degrees
// label: (*when pin is at the lock position,reset the output to deploy the stow pin*)
fb_rtrig_reset_deploy(CLK := (b_remote_on OR b_local_on) AND b_stow_pin_limit_lock); // R_TRIG
b_stow_pin_deploy R= fb_rtrig_reset_deploy.Q;
b_manual_stow R= fb_rtrig_reset_deploy.Q;
b_move_0_done R= fb_rtrig_reset_deploy.Q;
b_move_90_done R= fb_rtrig_reset_deploy.Q;
b_Horn R= fb_rtrig_reset_deploy.Q;
b_Alarm R= fb_rtrig_reset_deploy.Q;
b_stow_run R= fb_rtrig_reset_deploy.Q;
b_stow R= fb_rtrig_reset_deploy.Q;

// NETWORK 11
//   b_remote_on: in the remote mode
//   b_stow_pin_limit_unlock: the lock pin is at the lock position
//   b_stow_pin_retract: the command of stowing the antenna at 20_degrees
// label: (*when pin is at the unlock position,reset the output to retract the stow pin*)
fb_rtrig_reset_retract(CLK := (b_remote_on OR b_local_on) AND b_stow_pin_limit_unlock); // R_TRIG
b_stow_pin_retract R= fb_rtrig_reset_retract.Q;

// NETWORK 12

// NETWORK 13 (disabled)
//   b_remote_on: in the remote mode
//   b_limit_lock: the lock pin is at the lock position
//   b_scc_maintain: the command of stowing the antenna at 20_degrees
//   b_scc_stow: the command of stowing the antenna at 90_degrees
// label: (*when pin is at the lock position,reset the TCP command vlue*)
// rtrig_reset_TCP_lock(CLK := b_remote_on AND NOT b_limit_lock); // R_TRIG
// b_scc_maintain R= rtrig_reset_TCP_lock.Q;
// b_scc_stow R= rtrig_reset_TCP_lock.Q;

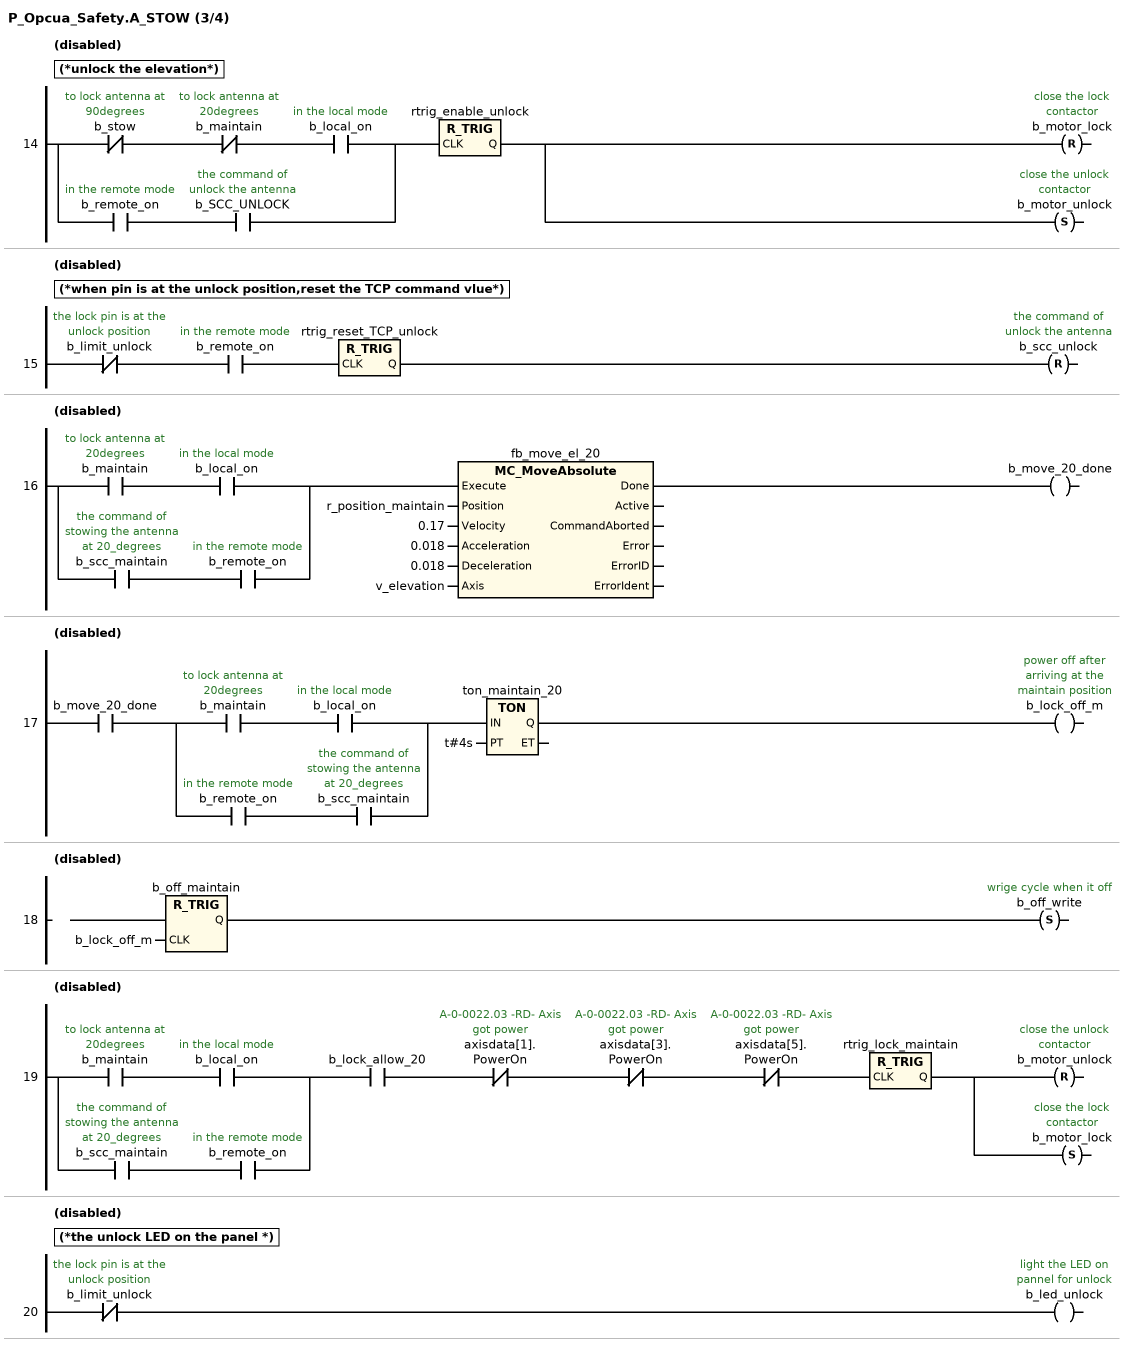
// NETWORK 14 (disabled)
//   b_stow: to lock antenna at 90degrees
//   b_maintain: to lock antenna at 20degrees
//   b_local_on: in the local mode
//   b_remote_on: in the remote mode
//   b_SCC_UNLOCK: the command of unlock the antenna
//   b_motor_lock: close the lock contactor
//   b_motor_unlock: close the unlock contactor
// label: (*unlock the elevation*)
// rtrig_enable_unlock(CLK := NOT b_stow AND NOT b_maintain AND b_local_on OR b_remote_on AND b_SCC_UNLOCK); // R_TRIG
// b_motor_lock R= rtrig_enable_unlock.Q;
// b_motor_unlock S= rtrig_enable_unlock.Q;

// NETWORK 15 (disabled)
//   b_limit_unlock: the lock pin is at the unlock position
//   b_remote_on: in the remote mode
//   b_scc_unlock: the command of unlock the antenna
// label: (*when pin is at the unlock position,reset the TCP command vlue*)
// rtrig_reset_TCP_unlock(CLK := NOT b_limit_unlock AND b_remote_on); // R_TRIG
// b_scc_unlock R= rtrig_reset_TCP_unlock.Q;

// NETWORK 16 (disabled)
//   b_maintain: to lock antenna at 20degrees
//   b_local_on: in the local mode
//   b_scc_maintain: the command of stowing the antenna at 20_degrees
//   b_remote_on: in the remote mode
//   v_elevation: Virtual axis "v_elevation" with axis number 8
// fb_move_el_20(
//     Execute := b_maintain AND b_local_on OR b_scc_maintain AND b_remote_on,
//     Position := r_position_maintain,
//     Velocity := 0.17,
//     Acceleration := 0.018,
//     Deceleration := 0.018,
//     Axis := v_elevation); // MC_MoveAbsolute
// b_move_20_done := fb_move_el_20.Done;

// NETWORK 17 (disabled)
//   b_maintain: to lock antenna at 20degrees
//   b_local_on: in the local mode
//   b_remote_on: in the remote mode
//   b_scc_maintain: the command of stowing the antenna at 20_degrees
//   b_lock_off_m: power off after arriving at the maintain position
// ton_maintain_20(IN := b_move_20_done AND (b_maintain AND b_local_on OR b_remote_on AND b_scc_maintain), PT := t#4s); // TON
// b_lock_off_m := ton_maintain_20.Q;

// NETWORK 18 (disabled)
//   b_lock_off_m: power off after arriving at the maintain position
//   b_off_write: wrige cycle when it off
// b_off_maintain(CLK := b_lock_off_m); // R_TRIG
// b_off_write S= b_off_maintain.Q;

// NETWORK 19 (disabled)
//   b_maintain: to lock antenna at 20degrees
//   b_local_on: in the local mode
//   b_scc_maintain: the command of stowing the antenna at 20_degrees
//   b_remote_on: in the remote mode
//   axisdata[1].PowerOn: A-0-0022.03 -RD- Axis got power
//   axisdata[3].PowerOn: A-0-0022.03 -RD- Axis got power
//   axisdata[5].PowerOn: A-0-0022.03 -RD- Axis got power
//   b_motor_unlock: close the unlock contactor
//   b_motor_lock: close the lock contactor
// rtrig_lock_maintain(CLK := (b_maintain AND b_local_on OR b_scc_maintain AND b_remote_on) AND b_lock_allow_20 AND NOT axisdata[1].PowerOn AND NOT axisdata[3].PowerOn AND NOT axisdata[5].PowerOn); // R_TRIG
// b_motor_unlock R= rtrig_lock_maintain.Q;
// b_motor_lock S= rtrig_lock_maintain.Q;

// NETWORK 20 (disabled)
//   b_limit_unlock: the lock pin is at the unlock position
//   b_led_unlock: light the LED on pannel for unlock
// label: (*the unlock LED on the panel *)
// b_led_unlock := NOT b_limit_unlock;

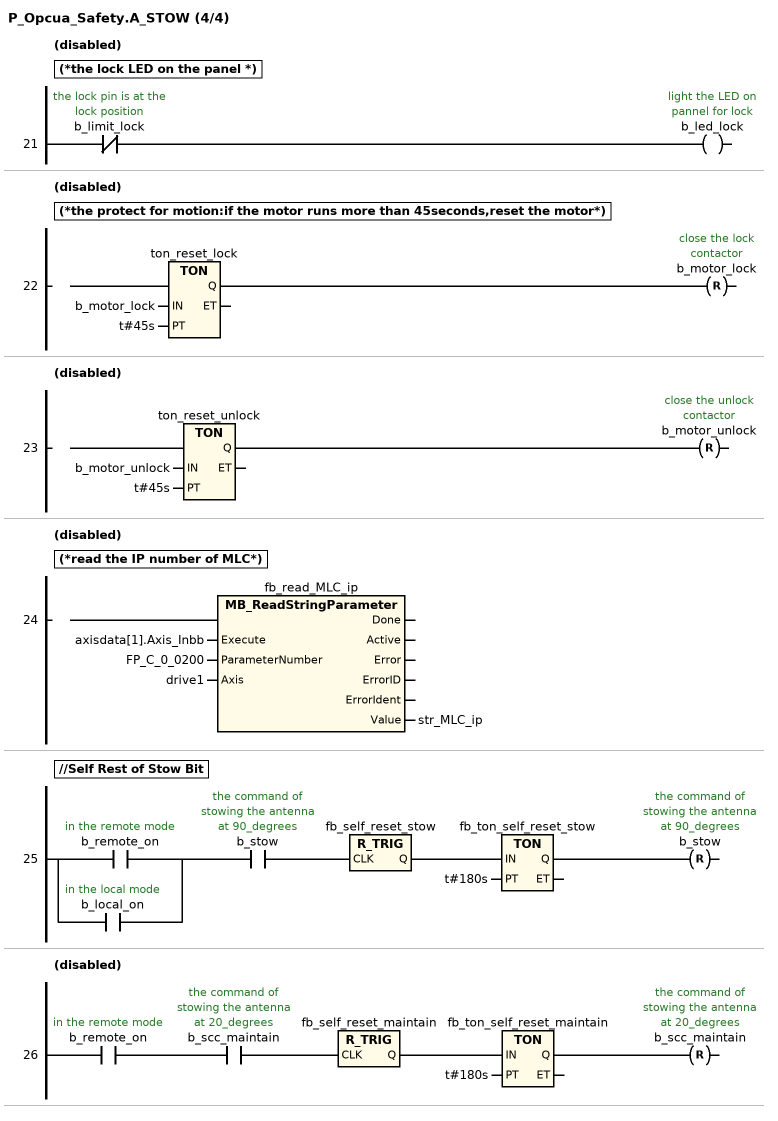
// NETWORK 21 (disabled)
//   b_limit_lock: the lock pin is at the lock position
//   b_led_lock: light the LED on pannel for lock
// label: (*the lock LED on the panel *)
// b_led_lock := NOT b_limit_lock;

// NETWORK 22 (disabled)
//   b_motor_lock: close the lock contactor
// label: (*the protect for motion:if the motor runs more than 45seconds,reset the motor*)
// ton_reset_lock(IN := b_motor_lock, PT := t#45s); // TON
// b_motor_lock R= ton_reset_lock.Q;

// NETWORK 23 (disabled)
//   b_motor_unlock: close the unlock contactor
// ton_reset_unlock(IN := b_motor_unlock, PT := t#45s); // TON
// b_motor_unlock R= ton_reset_unlock.Q;

// NETWORK 24 (disabled)
//   axisdata[1].Axis_Inbb: A-0-0021.13 -RD- Axis is ready for power to the amplifier (bb)
//   FP_C_0_0200: Engineering, IP address
//   drive1: Real axis "Drive1" with axis number 1
//   str_MLC_ip: IP number in MLC
// label: (*read the IP number of MLC*)
// fb_read_MLC_ip(
//     Execute := axisdata[1].Axis_Inbb,
//     ParameterNumber := FP_C_0_0200,
//     Axis := drive1,
//     Value => str_MLC_ip); // MB_ReadStringParameter

// NETWORK 25
//   b_remote_on: in the remote mode
//   b_local_on: in the local mode
//   b_stow: the command of stowing the antenna at 90_degrees
// label: //Self Rest of Stow Bit
fb_self_reset_stow(CLK := (b_remote_on OR b_local_on) AND b_stow); // R_TRIG
fb_ton_self_reset_stow(IN := fb_self_reset_stow.Q, PT := t#180s); // TON
b_stow R= fb_ton_self_reset_stow.Q;

// NETWORK 26 (disabled)
//   b_remote_on: in the remote mode
//   b_scc_maintain: the command of stowing the antenna at 20_degrees
// fb_self_reset_maintain(CLK := b_remote_on AND b_scc_maintain); // R_TRIG
// fb_ton_self_reset_maintain(IN := fb_self_reset_maintain.Q, PT := t#180s); // TON
// b_scc_maintain R= fb_ton_self_reset_maintain.Q;
END_ACTION

ACTION A_Interlock_Estop:
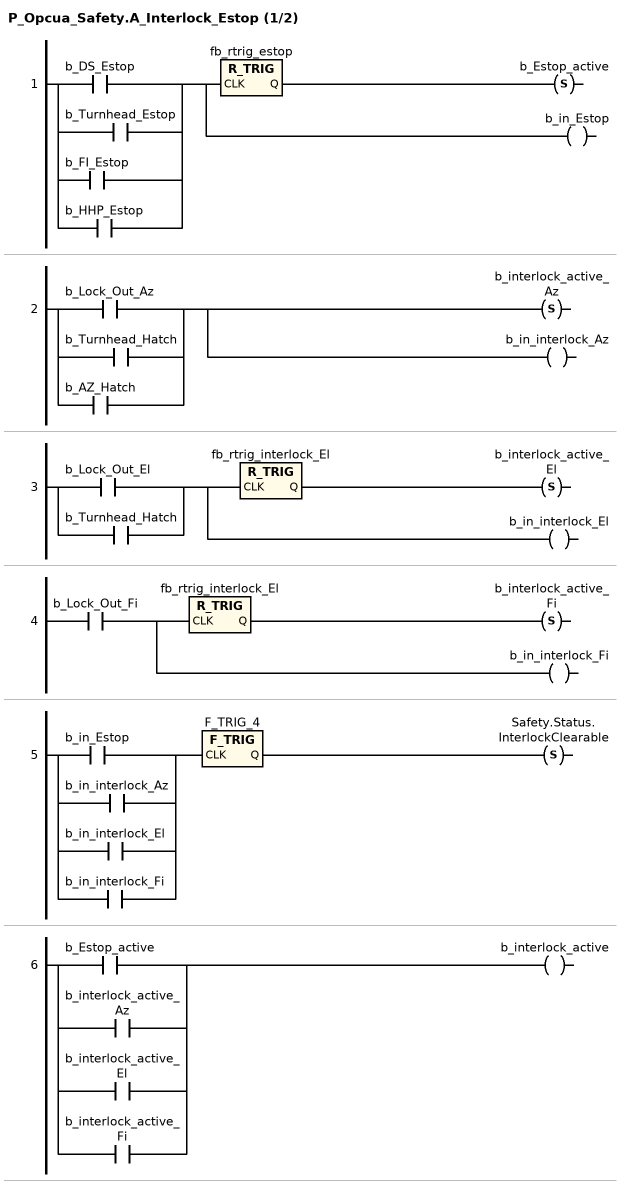
// NETWORK 1
_w3 := b_DS_Estop OR b_Turnhead_Estop OR b_FI_Estop OR b_HHP_Estop;
fb_rtrig_estop(CLK := _w3); // R_TRIG
b_Estop_active S= fb_rtrig_estop.Q;
b_in_Estop := _w3;

// NETWORK 2
_w4 := b_Lock_Out_Az OR b_Turnhead_Hatch OR b_AZ_Hatch;
b_interlock_active_Az S= _w4;
b_in_interlock_Az := _w4;

// NETWORK 3
_w5 := b_Lock_Out_El OR b_Turnhead_Hatch;
fb_rtrig_interlock_El(CLK := _w5); // R_TRIG
b_interlock_active_El S= fb_rtrig_interlock_El.Q;
b_in_interlock_El := _w5;

// NETWORK 4
fb_rtrig_interlock_El(CLK := b_Lock_Out_Fi); // R_TRIG
b_interlock_active_Fi S= fb_rtrig_interlock_El.Q;
b_in_interlock_Fi := b_Lock_Out_Fi;

// NETWORK 5
F_TRIG_4(CLK := b_in_Estop OR b_in_interlock_Az OR b_in_interlock_El OR b_in_interlock_Fi); // F_TRIG
Safety.Status.InterlockClearable S= F_TRIG_4.Q;

// NETWORK 6
b_interlock_active := b_Estop_active OR b_interlock_active_Az OR b_interlock_active_El OR b_interlock_active_Fi;

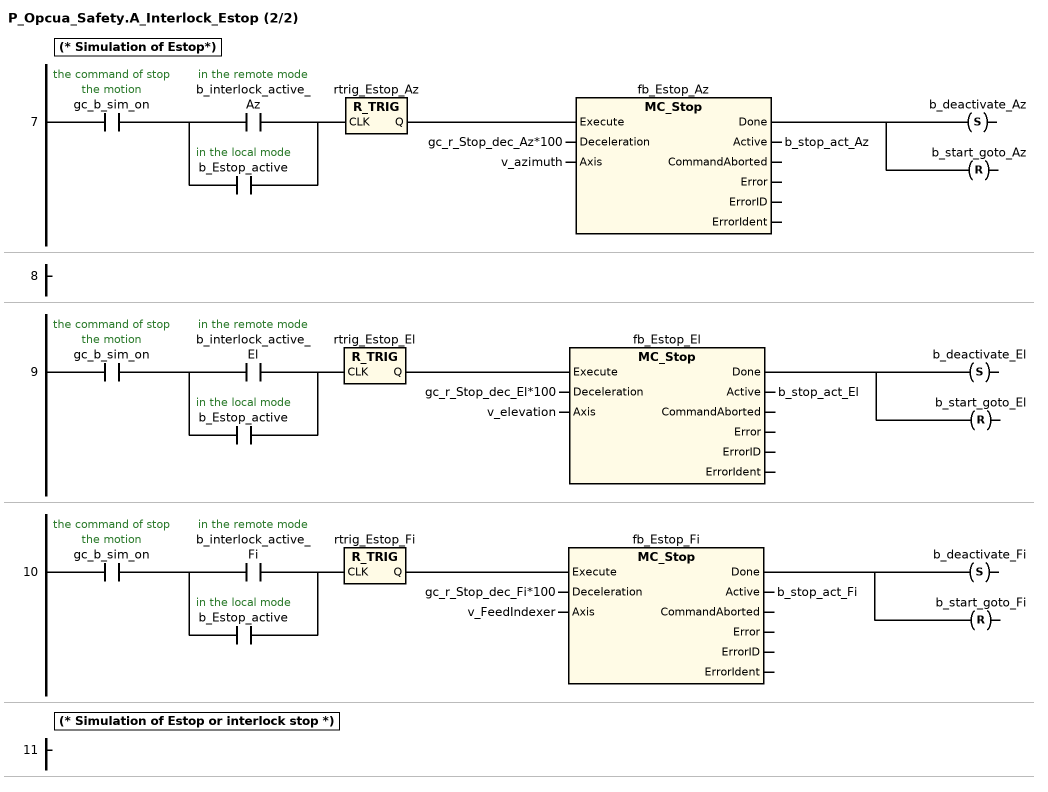
// NETWORK 7
//   gc_b_sim_on: the command of stop the motion
//   b_interlock_active_Az: in the remote mode
//   b_Estop_active: in the local mode
//   v_azimuth: Virtual axis "v_azimuth" with axis number 7
// label: (* Simulation of Estop*)
rtrig_Estop_Az(CLK := gc_b_sim_on AND (b_interlock_active_Az OR b_Estop_active)); // R_TRIG
fb_Estop_Az(
    Execute := rtrig_Estop_Az.Q,
    Deceleration := gc_r_Stop_dec_Az*100,
    Axis := v_azimuth,
    Active => b_stop_act_Az); // MC_Stop
b_deactivate_Az S= fb_Estop_Az.Done;
b_start_goto_Az R= fb_Estop_Az.Done;

// NETWORK 8

// NETWORK 9
//   gc_b_sim_on: the command of stop the motion
//   b_interlock_active_El: in the remote mode
//   b_Estop_active: in the local mode
//   v_elevation: Virtual axis "v_elevation" with axis number 8
rtrig_Estop_El(CLK := gc_b_sim_on AND (b_interlock_active_El OR b_Estop_active)); // R_TRIG
fb_Estop_El(
    Execute := rtrig_Estop_El.Q,
    Deceleration := gc_r_Stop_dec_El*100,
    Axis := v_elevation,
    Active => b_stop_act_El); // MC_Stop
b_deactivate_El S= fb_Estop_El.Done;
b_start_goto_El R= fb_Estop_El.Done;

// NETWORK 10
//   gc_b_sim_on: the command of stop the motion
//   b_interlock_active_Fi: in the remote mode
//   b_Estop_active: in the local mode
//   v_FeedIndexer: Virtual axis "v_polarization" with axis number 9
rtrig_Estop_Fi(CLK := gc_b_sim_on AND (b_interlock_active_Fi OR b_Estop_active)); // R_TRIG
fb_Estop_Fi(
    Execute := rtrig_Estop_Fi.Q,
    Deceleration := gc_r_Stop_dec_Fi*100,
    Axis := v_FeedIndexer,
    Active => b_stop_act_Fi); // MC_Stop
b_deactivate_Fi S= fb_Estop_Fi.Done;
b_start_goto_Fi R= fb_Estop_Fi.Done;

// NETWORK 11
// label: (* Simulation of Estop or interlock stop *)
END_ACTION

END_PROGRAM

// IndraMotionMlc1/Application/POUs/OPCUA/OPCUA_Node/P_Opcua_CommandArbiter
PROGRAM P_Opcua_CommandArbiter
VAR
	cmds: CmdResponseType;
END_VAR

CommandArbiter();
//CommandArbiter.Status.DscCmdAuthority;


(* if hhp connected then 
    CommandArbiter.DscCmdAuthority:= HHP;
	End *)

END_PROGRAM

// IndraMotionMlc1/Application/POUs/OPCUA/OPCUA_Node/P_Opcua_Time_cds
PROGRAM P_Opcua_Time_cds
VAR
	IL_SysTime64_0: IL_SysTime64;
	Current_time: SYS_TIME64;
	UnixSeconds: Lreal;
	i_num_quarter_test: DINT;
	current_time_pos_test: LREAL;
	lr_MJD_Test: LREAL;
	
	dummy: Lreal;
	dummy2: Bool;
END_VAR

Time_cds();

P_Opcua_Time_cds.Get_Time();
//Time_cds.Status.TAIOffset:=Current_time.HighValue*65536+Current_time.LowValue;
//Calculate TAI offset 
//Time_cds.Status.TAIOffset:=Current_time.HighValue*65536+Current_time.LowValue;
//Time_cds.Status.TAIOffset:=((Current_time.HighValue+4294967295)/1000000+ Current_time.LowValue/1000000);
UnixSeconds:=(TO_LREAL(Current_time.HighValue)*4294967295+TO_LREAL(Current_time.LowValue))/1000000; //UTC 
//Time_cds.Status.TAIOffset:=UnixSeconds-UnixToSKAEpoch-(Time_cds.Status.LeapSecPTP-Time_cds.Status.UTCtoSkaoEpochSec);

lr_MJD_Test:= UnixSeconds/86400+40587;

 // This should be the TAI offset after the SKAO epoch. The time from the Time Virtual axis.
//Time_cds.Status.DscTimeSyncSource:=Source_Timesync;

Time_cds.Status.LeapSecPTP:=LeapSecPTP;   
IF Source_Timesync = DscTimeSyncSourceType.PTP THEN
	Time_cds.Status.TimeSourceAddrNTP:=IP_Adress_PTP;
ELSIF Source_Timesync = DscTimeSyncSourceType.NTP THEN
	Time_cds.Status.TimeSourceAddrNTP:=IP_Adress_NTP;
ELSE
	Time_cds.Status.TimeSourceAddrNTP:=str_MLC_ip;
END_IF

IF Source_Timesync = DscTimeSyncSourceType.PTP THEN
	Time_cds.Status.TimeSynced:=b_M_time_done;
	b_no_SetDateTime:=FALSE;
ELSIF Source_Timesync = DscTimeSyncSourceType.NTP THEN
	//Time_cds.Status.TimeSynced:=b_M_time_done;
	b_no_SetDateTime:=FALSE;
ELSE
	
    Time_cds.Status.TimeSynced:=b_M_time_done;
	// need to use system time to calculate MJD
	b_no_SetDateTime:=TRUE;
	
	di_MJD_day := LREAL_TO_DINT(TRUNC(UnixSeconds/86400+40587));
	i_num_quarter:=TRUNC((UnixSeconds-DINT_TO_LREAL(TRUNC(UnixSeconds/86400)*86400))/360);
	current_time_pos_test:=UnixSeconds-DINT_TO_LREAL(TRUNC(UnixSeconds/86400)*86400)-i_num_quarter*360;
	dummy:=P_UDP_To_NTP.current_time_pos-current_time_pos_test;
	dummy2:=(ABS(dummy)>=0.10);
	IF (ABS(dummy)>=0.10 AND NOT(b_track_on)) THEN
		P_UDP_To_NTP.current_time_pos:=current_time_pos_test;
	   	P_UDP_To_NTP.b_NTP_set_up:=TRUE;
	ELSE 
		P_UDP_To_NTP.b_NTP_set_up:=FALSE;	
	
	END_IF
	
	
	
END_IF

ACTION Get_Time:
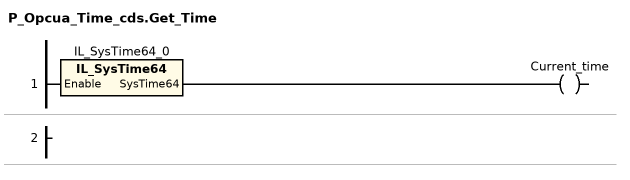
// NETWORK 1
IL_SysTime64_0(Enable := TRUE); // IL_SysTime64
Current_time := IL_SysTime64_0.SysTime64;

// NETWORK 2
END_ACTION

END_PROGRAM

// IndraMotionMlc1/Application/POUs/OPCUA/OPCUA_Node/P_Opcua_Management
PROGRAM P_Opcua_Management
VAR
	R_total_distance_AZ_old:LREAL;
	R_total_distance_EL_deg_old:LREAL;
	R_total_distance_EL_m_old:LREAL;
	R_total_distance_FI_old:LREAL;
	count_i:UINT;
	(*<<<<<<<<<<<<<<<<<<<<<<<<<<<<<<<<<<<< Stop >>>>>>>>>>>>>>>>>>>>>>>>>>>>>*)
	b_stop_Az_done: BOOL;
	b_stop_El_done: BOOL;
	b_stop_Fi_done: BOOL;
	fb_stop_Az: MC_Stop;
	fb_stop_El: MC_Stop;
	fb_stop_Fi: MC_Stop;
	rtrig_stop_Az: R_TRIG;
	rtrig_stop_El: R_TRIG;
	rtrig_stop_Fi: R_TRIG;
	rtrig_stop_stow: R_TRIG;
	rtrig_reset_stop: R_TRIG;
	
	(*<<<<<<<<<<<<<<<<<<<<<<<<<<<<<<<<<<<< Goto >>>>>>>>>>>>>>>>>>>>>>>>>>>>>*)
	// Az
	
	b_goto_done_Az: BOOL;
	b_active_Az:     BOOL;
	b_moving_Az: BOOL;
	fb_goto_Az: MC_MoveRelative;
	fb_start_goto_Az: R_Trig;
	fb_goto_done_Az : R_Trig;
	
	// El
	
	b_goto_done_El: BOOL;
	b_active_El:     BOOL;
	b_moving_El: BOOL;
	fb_goto_El: MC_MoveRelative;
	fb_start_goto_El: R_Trig;
	fb_goto_done_El : R_Trig;
	//Fi
	b_goto_done_Fi: BOOL;
	b_active_Fi:     BOOL;
	b_moving_Fi: BOOL;
	fb_goto_Fi: MC_MoveRelative;
	fb_start_goto_Fi: R_Trig;
	fb_goto_done_Fi : R_Trig;
	
(*<<<<<<<<<<<<<<<<<<<<<<<<<<<<<<<<<<<<<<<<<<<<<<<<<<<power>>>>>>>>>>>>>>>>>>>>>>>>>>>>>>>>>>>>*)
	ton_pow_off_Az: TON;
	ton_pow_off_El: TON;
	ton_pow_off_Fi: TON;
	rtrig_power_Az: R_TRIG;
	rtrig_power_El: R_TRIG;
	rtrig_power_Fi: R_TRIG;
	fb_ton_El: TON;
	fb_ton_Fi: TON;
	rtrig_off_Az: R_TRIG;
	rtrig_off_El: R_TRIG;
	rtrig_off_Fi: R_TRIG;
	rtrig_power_power: R_TRIG;
	b_pwr_on:BOOL;
	b_pwr_off: BOOL;
	b_clear_off_done_Az1: BOOL;
	b_clear_off_done_Az2: BOOL;
	b_clear_off_done_El: BOOL;
	b_clear_off_done_Fi1: BOOL;
	b_clear_off_done_Fi2: BOOL;
	
	FB_clear_error_off_Az1:MB_WriteParameter;
	FB_clear_error_off_Az2:MB_WriteParameter;
	FB_clear_error_off_El:MB_WriteParameter;
	FB_clear_error_off_Fi1:MB_WriteParameter;
	FB_clear_error_off_Fi2:MB_WriteParameter;
	rtrig_err: R_TRIG;
	rtrig_clear_done: R_TRIG;
	fb_ton_stow: TON;
	
	fb_rtrig_stow_deactivate1: R_TRIG;
	fb_rtrig_stow_deactivate: R_TRIG;
	b_execute_goto_Az: BOOL;
	R_TRIG_0: R_TRIG;
	R_TRIG_1: R_TRIG;
	rtrig_stop_goto_el: R_TRIG;
	rtrig_stop_goto_az: R_TRIG;
	fb_TON_2: TON;
	fb_TON_1: TON;
	r_goto_Az_rel: REAL;
	r_goto_El_rel: LREAL;
	r_goto_fi_rel: LREAL;
END_VAR
VAR // added by the converter: edge detectors and wires of the graphical bodies
    _w1, _w2 : BOOL;
END_VAR


(***********Management.DscState***********)
IF azimuth.Status.AxisState=axisstatetype.StartUp OR elevation.Status.AxisState=axisstatetype.StartUp THEN
	Management.Status.DscState:=DscstateType.StartUp;
END_IF

IF azimuth.Status.AxisState=axisstatetype.Standby AND elevation.Status.AxisState=axisstatetype.Standby THEN
	Management.Status.DscState:=DscstateType.Standby;
END_IF

IF azimuth.Status.AxisState=axisstatetype.Activating OR elevation.Status.AxisState=axisstatetype.Activating THEN
	Management.Status.DscState:=DscstateType.Activating;
END_IF

IF azimuth.Status.AxisState=axisstatetype.Deactivating OR elevation.Status.AxisState=axisstatetype.Deactivating THEN
	Management.Status.DscState:=DscstateType.Deactivating;
END_IF

IF azimuth.Status.AxisState=axisstatetype.Standstill OR elevation.Status.AxisState=axisstatetype.Standstill THEN
	Management.Status.DscState:=DscstateType.Standstill;
END_IF

IF azimuth.Status.AxisState=axisstatetype.Stopping OR elevation.Status.AxisState=axisstatetype.Stopping THEN
	Management.Status.DscState:=DscstateType.stopping;
END_IF

IF azimuth.Status.AxisState=axisstatetype.Jog OR elevation.Status.AxisState=axisstatetype.Jog THEN
	Management.Status.DscState:=DscstateType.Jog;
END_IF

IF azimuth.Status.AxisState=axisstatetype.Slew OR elevation.Status.AxisState=axisstatetype.Slew THEN //capitalise S in slew
	Management.Status.DscState:=DscstateType.slew;
END_IF

IF azimuth.Status.AxisState=axisstatetype.Track AND elevation.Status.AxisState=axisstatetype.Track THEN
	Management.Status.DscState:=DscstateType.Track;
END_IF

IF azimuth.Status.AxisState=axisstatetype.Stowed THEN
	Management.Status.DscState:=DscstateType.Stowed;
END_IF
IF azimuth.Status.AxisState=axisstatetype.Locked OR elevation.Status.AxisState=axisstatetype.Locked THEN
	Management.Status.DscState:=DscstateType.Locked;
END_IF

IF azimuth.Status.AxisState=axisstatetype.Locked_Stowed OR elevation.Status.AxisState=axisstatetype.Locked_Stowed THEN
	Management.Status.DscState:=DscstateType.Locked_Stowed;
END_IF

// This one isn't going to work 
IF b_stow_pin_limit_lock AND (azimuth.Status.AxisState=axisstatetype.Locked OR elevation.Status.AxisState=axisstatetype.Locked) THEN     // Need to check Errors and interlocks to go into locked
	Management.Status.DscState:=DscstateType.Locked_Stowed;
END_IF

(*IF b_in_Estop THEN
	Management.Status.DscState:=DscstateType.Locked;  //Axis also need to go into locked state
END_IF
*)


// Work out where FiPOS is 
IF b_goto_done_Fi THEN 
	IF r_pos_fi_v < gc_r_band_optical+gc_r_band_tolerance AND r_pos_fi_v > gc_r_band_optical-gc_r_band_tolerance THEN 
		Management.Status.FiPos:= bandtype.Optical;
	ELSIF
		r_pos_fi_v < gc_r_band_1+gc_r_band_tolerance AND r_pos_fi_v > gc_r_band_1-gc_r_band_tolerance THEN 
		Management.Status.FiPos:= bandtype.Band_1;
	ELSIF
		r_pos_fi_v < gc_r_band_2+gc_r_band_tolerance AND r_pos_fi_v > gc_r_band_2-gc_r_band_tolerance THEN 
		Management.Status.FiPos:= bandtype.Band_2;
	ELSIF
		r_pos_fi_v < gc_r_band_3+gc_r_band_tolerance AND r_pos_fi_v > gc_r_band_3-gc_r_band_tolerance THEN 
		Management.Status.FiPos:= bandtype.Band_3;
	ELSIF
		r_pos_fi_v < gc_r_band_4+gc_r_band_tolerance AND r_pos_fi_v > gc_r_band_4-gc_r_band_tolerance THEN 
		Management.Status.FiPos:= bandtype.Band_4;
	ELSIF
		r_pos_fi_v < gc_r_band_5a+gc_r_band_tolerance AND r_pos_fi_v > gc_r_band_5a-gc_r_band_tolerance THEN 
		Management.Status.FiPos:= bandtype.Band_5a;
	ELSIF
		r_pos_fi_v < gc_r_band_5b+gc_r_band_tolerance AND r_pos_fi_v > gc_r_band_5b-gc_r_band_tolerance THEN 
		Management.Status.FiPos:= bandtype.Band_5b;
	ELSIF
		r_pos_fi_v < gc_r_band_6+gc_r_band_tolerance AND r_pos_fi_v > gc_r_band_6-gc_r_band_tolerance THEN 
		Management.Status.FiPos:= bandtype.Band_6;
	ELSE
		Management.Status.FiPos:= bandtype.Unknown;
	END_IF

END_IF


